LIN {X 0.038,Y -348.064,Z 1859.529,A 0.000,B 0.000,C 90.000,E1 275.163} C_DIS
LIN {X -0.149,Y -343.133,Z 1859.525,A 0.000,B 0.000,C 90.000,E1 274.588} C_DIS
LIN {X 0.037,Y -337.603,Z 1859.522,A 0.000,B 0.000,C 90.000,E1 273.955} C_DIS
LIN {X 0.034,Y -331.682,Z 1859.519,A 0.000,B 0.000,C 90.000,E1 273.383} C_DIS
LIN {X -0.019,Y -325.520,Z 1859.516,A 0.000,B 0.000,C 90.000,E1 272.865} C_DIS
LIN {X -0.139,Y -319.108,Z 1859.513,A 0.000,B 0.000,C 90.000,E1 272.407} C_DIS
LIN {X 0.029,Y -312.422,Z 1859.511,A 0.000,B 0.000,C 90.000,E1 271.949} C_DIS
LIN {X -0.128,Y -305.605,Z 1859.509,A 0.000,B 0.000,C 90.000,E1 271.604} C_DIS
LIN {X 0.010,Y -298.212,Z 1859.507,A 0.000,B 0.000,C 90.000,E1 271.260} C_DIS
LIN {X -0.113,Y -290.603,Z 1859.506,A 0.000,B 0.000,C 90.000,E1 271.031} C_DIS
LIN {X 0.034,Y -283.001,Z 1859.505,A 0.000,B 0.000,C 90.000,E1 270.802} C_DIS
LIN {X -0.029,Y -268.014,Z 1859.503,A 0.000,B 0.000,C 90.000,E1 270.516} C_DIS
LIN {X -0.049,Y -246.564,Z 1859.501,A 0.000,B 0.000,C 90.000,E1 270.115} C_DIS
LIN {X -0.031,Y -234.364,Z 1859.500,A 0.000,B 0.000,C 90.000,E1 269.943} C_DIS
LIN {X 0.025,Y -226.280,Z 1859.499,A 0.000,B 0.000,C 90.000,E1 269.885} C_DIS
LIN {X 0.000,Y -181.539,Z 1859.499,A 0.000,B 0.000,C 90.000,E1 269.885} C_DIS
LIN {X -0.082,Y -180.788,Z 1859.471,A 0.000,B 0.000,C 90.000,E1 264.780} C_DIS
LIN {X -0.008,Y -178.886,Z 1859.443,A 0.000,B 0.000,C 90.000,E1 259.690} C_DIS
LIN {X 0.067,Y -175.929,Z 1859.414,A 0.000,B 0.000,C 90.000,E1 254.574} C_DIS
LIN {X 0.013,Y -175.371,Z 1859.410,A 0.000,B 0.000,C 90.000,E1 253.740} C_DIS
LIN {X 0.072,Y -172.148,Z 1859.386,A 0.000,B 0.000,C 90.000,E1 249.444} C_DIS
LIN {X 0.048,Y -171.613,Z 1859.381,A 0.000,B 0.000,C 90.000,E1 248.592} C_DIS
LIN {X 0.036,Y -167.835,Z 1859.357,A 0.000,B 0.000,C 90.000,E1 244.280} C_DIS
LIN {X 0.054,Y -166.562,Z 1859.348,A 0.000,B 0.000,C 90.000,E1 242.538} C_DIS
LIN {X -0.036,Y -162.556,Z 1859.323,A 0.000,B 0.000,C 90.000,E1 238.201} C_DIS
LIN {X 0.023,Y -161.235,Z 1859.313,A 0.000,B 0.000,C 90.000,E1 236.421} C_DIS
LIN {X 0.058,Y -157.240,Z 1859.289,A 0.000,B 0.000,C 90.000,E1 231.984} C_DIS
LIN {X -0.019,Y -155.963,Z 1859.279,A 0.000,B 0.000,C 90.000,E1 230.231} C_DIS
LIN {X 0.039,Y -152.218,Z 1859.254,A 0.000,B 0.000,C 90.000,E1 225.729} C_DIS
LIN {X 0.060,Y -150.462,Z 1859.239,A 0.000,B 0.000,C 90.000,E1 223.014} C_DIS
LIN {X 0.086,Y -147.187,Z 1859.214,A 0.000,B 0.000,C 90.000,E1 218.463} C_DIS
LIN {X 0.052,Y -145.205,Z 1859.194,A 0.000,B 0.000,C 90.000,E1 214.818} C_DIS
LIN {X -0.038,Y -142.340,Z 1859.163,A 0.000,B 0.000,C 90.000,E1 209.333} C_DIS
LIN {X 0.016,Y -141.729,Z 1859.153,A 0.000,B 0.000,C 90.000,E1 207.462} C_DIS
LIN {X -0.003,Y -139.482,Z 1859.116,A 0.000,B 0.000,C 90.000,E1 200.972} C_DIS
LIN {X -0.014,Y -138.980,Z 1859.101,A 0.000,B 0.000,C 90.000,E1 198.181} C_DIS
LIN {X -0.053,Y -138.332,Z 1859.054,A 0.000,B 0.000,C 90.000,E1 189.792} C_DIS
LIN {X -0.028,Y -139.427,Z 1859.008,A 0.000,B 0.000,C 90.000,E1 181.375} C_DIS
LIN {X 0.025,Y -141.354,Z 1858.971,A 0.000,B 0.000,C 90.000,E1 174.837} C_DIS
LIN {X 0.002,Y -142.707,Z 1858.956,A 0.000,B 0.000,C 90.000,E1 172.064} C_DIS
LIN {X -0.040,Y -145.081,Z 1858.930,A 0.000,B 0.000,C 90.000,E1 167.465} C_DIS
LIN {X -0.044,Y -147.706,Z 1858.910,A 0.000,B 0.000,C 90.000,E1 163.795} C_DIS
LIN {X 0.040,Y -150.359,Z 1858.890,A 0.000,B 0.000,C 90.000,E1 160.115} C_DIS
LIN {X 0.058,Y -153.784,Z 1858.870,A 0.000,B 0.000,C 90.000,E1 156.485} C_DIS
LIN {X -0.021,Y -157.197,Z 1858.849,A 0.000,B 0.000,C 90.000,E1 152.922} C_DIS
LIN {X 0.060,Y -161.358,Z 1858.830,A 0.000,B 0.000,C 90.000,E1 149.331} C_DIS
LIN {X 0.072,Y -165.561,Z 1858.810,A 0.000,B 0.000,C 90.000,E1 145.801} C_DIS
LIN {X -0.044,Y -170.477,Z 1858.791,A 0.000,B 0.000,C 90.000,E1 142.351} C_DIS
LIN {X 0.105,Y -175.358,Z 1858.772,A 0.000,B 0.000,C 90.000,E1 138.852} C_DIS
LIN {X -0.032,Y -180.982,Z 1858.753,A 0.000,B 0.000,C 90.000,E1 135.486} C_DIS
LIN {X -0.045,Y -186.408,Z 1858.734,A 0.000,B 0.000,C 90.000,E1 132.123} C_DIS
LIN {X -0.106,Y -191.036,Z 1858.720,A 0.000,B 0.000,C 90.000,E1 129.644} C_DIS
LIN {X 0.086,Y -196.818,Z 1858.702,A 0.000,B 0.000,C 90.000,E1 126.297} C_DIS
LIN {X 0.005,Y -200.073,Z 1858.693,A 0.000,B 0.000,C 90.000,E1 124.692} C_DIS
LIN {X -0.001,Y -207.572,Z 1858.670,A 0.000,B 0.000,C 90.000,E1 120.669} C_DIS
LIN {X 0.002,Y -210.778,Z 1858.661,A 0.000,B 0.000,C 90.000,E1 119.077} C_DIS
LIN {X 0.010,Y -216.622,Z 1858.644,A 0.000,B 0.000,C 90.000,E1 115.924} C_DIS
LIN {X -0.080,Y -219.706,Z 1858.635,A 0.000,B 0.000,C 90.000,E1 114.387} C_DIS
LIN {X 0.069,Y -224.078,Z 1858.621,A 0.000,B 0.000,C 90.000,E1 111.844} C_DIS
LIN {X 0.051,Y -283.399,Z 1858.621,A 0.000,B 0.000,C 90.000,E1 111.844} C_DIS
LIN {X 0.136,Y -286.194,Z 1858.621,A 0.000,B 0.000,C 90.000,E1 111.770} C_DIS
LIN {X 0.002,Y -290.672,Z 1858.620,A 0.000,B 0.000,C 90.000,E1 111.535} C_DIS
LIN {X -0.029,Y -293.267,Z 1858.618,A 0.000,B 0.000,C 90.000,E1 111.280} C_DIS
LIN {X -0.184,Y -297.015,Z 1858.615,A 0.000,B 0.000,C 90.000,E1 110.737} C_DIS
LIN {X 0.111,Y -310.328,Z 1858.602,A 0.000,B 0.000,C 90.000,E1 108.362} C_DIS
LIN {X -0.076,Y -325.008,Z 1858.590,A 0.000,B 0.000,C 90.000,E1 106.134} C_DIS
LIN {X -0.094,Y -338.778,Z 1858.579,A 0.000,B 0.000,C 90.000,E1 104.245} C_DIS
LIN {X 0.162,Y -353.741,Z 1858.569,A 0.000,B 0.000,C 90.000,E1 102.355} C_DIS
LIN {X -0.081,Y -372.155,Z 1858.557,A 0.000,B 0.000,C 90.000,E1 100.366} C_DIS
LIN {X -0.019,Y -391.045,Z 1858.547,A 0.000,B 0.000,C 90.000,E1 98.511} C_DIS
LIN {X -0.022,Y -410.274,Z 1858.538,A 0.000,B 0.000,C 90.000,E1 96.834} C_DIS
LIN {X -0.127,Y -432.668,Z 1858.528,A 0.000,B 0.000,C 90.000,E1 95.106} C_DIS
LIN {X -0.159,Y -438.325,Z 1858.526,A 0.000,B 0.000,C 90.000,E1 94.702} C_DIS
LIN {X 0.046,Y -440.785,Z 1858.525,A 0.000,B 0.000,C 90.000,E1 94.473} C_DIS
LIN {X 0.181,Y -444.365,Z 1858.522,A 0.000,B 0.000,C 90.000,E1 94.012} C_DIS
LIN {X -0.093,Y -445.799,Z 1858.521,A 0.000,B 0.000,C 90.000,E1 93.784} C_DIS
LIN {X 0.079,Y -446.874,Z 1858.520,A 0.000,B 0.000,C 90.000,E1 93.498} C_DIS
LIN {X 0.033,Y -448.156,Z 1858.517,A 0.000,B 0.000,C 90.000,E1 92.980} C_DIS
LIN {X -0.029,Y -448.461,Z 1858.514,A 0.000,B 0.000,C 90.000,E1 92.465} C_DIS
LIN {X -0.082,Y -447.838,Z 1858.511,A 0.000,B 0.000,C 90.000,E1 91.949} C_DIS
LIN {X -0.118,Y -446.196,Z 1858.508,A 0.000,B 0.000,C 90.000,E1 91.432} C_DIS
LIN {X 0.078,Y -444.907,Z 1858.506,A 0.000,B 0.000,C 90.000,E1 91.146} C_DIS
LIN {X 0.008,Y -433.406,Z 1858.496,A 0.000,B 0.000,C 90.000,E1 89.312} C_DIS
LIN {X 0.020,Y -423.403,Z 1858.487,A 0.000,B 0.000,C 90.000,E1 87.707} C_DIS
LIN {X -0.030,Y -411.622,Z 1858.477,A 0.000,B 0.000,C 90.000,E1 85.812} C_DIS
LIN {X 0.122,Y -399.742,Z 1858.466,A 0.000,B 0.000,C 90.000,E1 83.856} C_DIS
LIN {X 0.057,Y -387.787,Z 1858.455,A 0.000,B 0.000,C 90.000,E1 81.894} C_DIS
LIN {X -0.131,Y -375.877,Z 1858.444,A 0.000,B 0.000,C 90.000,E1 79.916} C_DIS
LIN {X 0.121,Y -357.712,Z 1858.426,A 0.000,B 0.000,C 90.000,E1 76.645} C_DIS
LIN {X 0.086,Y -342.275,Z 1858.409,A 0.000,B 0.000,C 90.000,E1 73.630} C_DIS
LIN {X 0.140,Y -330.364,Z 1858.395,A 0.000,B 0.000,C 90.000,E1 71.148} C_DIS
LIN {X 0.027,Y -318.726,Z 1858.381,A 0.000,B 0.000,C 90.000,E1 68.646} C_DIS
LIN {X 0.063,Y -306.241,Z 1858.365,A 0.000,B 0.000,C 90.000,E1 65.741} C_DIS
LIN {X -0.036,Y -296.668,Z 1858.353,A 0.000,B 0.000,C 90.000,E1 63.461} C_DIS
LIN {X -0.088,Y -285.985,Z 1858.338,A 0.000,B 0.000,C 90.000,E1 60.795} C_DIS
LIN {X -0.072,Y -276.568,Z 1858.324,A 0.000,B 0.000,C 90.000,E1 58.408} C_DIS
LIN {X 0.019,Y -267.105,Z 1858.311,A 0.000,B 0.000,C 90.000,E1 55.960} C_DIS
LIN {X -0.016,Y -257.528,Z 1858.297,A 0.000,B 0.000,C 90.000,E1 53.497} C_DIS
LIN {X 0.042,Y -247.918,Z 1858.283,A 0.000,B 0.000,C 90.000,E1 50.964} C_DIS
LIN {X -0.008,Y -237.078,Z 1858.267,A 0.000,B 0.000,C 90.000,E1 48.038} C_DIS
LIN {X -0.084,Y -225.302,Z 1858.248,A 0.000,B 0.000,C 90.000,E1 44.676} C_DIS
LIN {X -0.007,Y -214.152,Z 1858.229,A 0.000,B 0.000,C 90.000,E1 41.191} C_DIS
LIN {X -0.087,Y -206.142,Z 1858.214,A 0.000,B 0.000,C 90.000,E1 38.463} C_DIS
LIN {X 0.038,Y -197.835,Z 1858.196,A 0.000,B 0.000,C 90.000,E1 35.231} C_DIS
LIN {X -0.051,Y -190.265,Z 1858.178,A 0.000,B 0.000,C 90.000,E1 32.005} C_DIS
LIN {X -0.032,Y -183.427,Z 1858.159,A 0.000,B 0.000,C 90.000,E1 28.693} C_DIS
LIN {X -0.033,Y -177.257,Z 1858.141,A 0.000,B 0.000,C 90.000,E1 25.335} C_DIS
LIN {X 0.065,Y -171.918,Z 1858.122,A 0.000,B 0.000,C 90.000,E1 21.897} C_DIS
LIN {X -0.053,Y -167.341,Z 1858.103,A 0.000,B 0.000,C 90.000,E1 18.489} C_DIS
LIN {X -0.063,Y -163.572,Z 1858.083,A 0.000,B 0.000,C 90.000,E1 15.009} C_DIS
LIN {X 0.033,Y -161.193,Z 1858.069,A 0.000,B 0.000,C 90.000,E1 12.355} C_DIS
LIN {X 0.014,Y -161.371,Z 1858.069,A 0.000,B 0.000,C 90.000,E1 12.355} C_DIS
LIN {X -0.062,Y -168.654,Z 1858.067,A 0.000,B 0.000,C 90.000,E1 12.119} C_DIS
LIN {X -0.066,Y -173.315,Z 1858.066,A 0.000,B 0.000,C 90.000,E1 11.883} C_DIS
LIN {X 0.008,Y -174.617,Z 1858.064,A 0.000,B 0.000,C 90.000,E1 11.535} C_DIS
LIN {X 0.065,Y -176.312,Z 1858.059,A 0.000,B 0.000,C 90.000,E1 10.658} C_DIS
LIN {X -0.076,Y -177.310,Z 1858.055,A 0.000,B 0.000,C 90.000,E1 9.849} C_DIS
LIN {X 0.051,Y -178.596,Z 1858.045,A 0.000,B 0.000,C 90.000,E1 8.106} C_DIS
LIN {X 0.036,Y -179.856,Z 1858.031,A 0.000,B 0.000,C 90.000,E1 5.568} C_DIS
LIN {X 0.071,Y -181.214,Z 1858.012,A 0.000,B 0.000,C 90.000,E1 2.178} C_DIS
LIN {X 0.026,Y -182.550,Z 1857.993,A 0.000,B 0.000,C 90.000,E1 358.682} C_DIS
LIN {X 0.018,Y -184.224,Z 1857.969,A 0.000,B 0.000,C 90.000,E1 354.489} C_DIS
LIN {X -0.049,Y -186.005,Z 1857.946,A 0.000,B 0.000,C 90.000,E1 350.330} C_DIS
LIN {X -0.063,Y -187.969,Z 1857.923,A 0.000,B 0.000,C 90.000,E1 346.172} C_DIS
LIN {X 0.031,Y -190.042,Z 1857.900,A 0.000,B 0.000,C 90.000,E1 342.000} C_DIS
LIN {X -0.052,Y -192.174,Z 1857.877,A 0.000,B 0.000,C 90.000,E1 337.901} C_DIS
LIN {X 0.044,Y -194.600,Z 1857.854,A 0.000,B 0.000,C 90.000,E1 333.768} C_DIS
LIN {X 0.120,Y -197.468,Z 1857.832,A 0.000,B 0.000,C 90.000,E1 329.665} C_DIS
LIN {X -0.100,Y -200.742,Z 1857.809,A 0.000,B 0.000,C 90.000,E1 325.674} C_DIS
LIN {X 0.014,Y -204.489,Z 1857.787,A 0.000,B 0.000,C 90.000,E1 321.618} C_DIS
LIN {X -0.012,Y -208.970,Z 1857.765,A 0.000,B 0.000,C 90.000,E1 317.634} C_DIS
LIN {X 0.044,Y -212.502,Z 1857.751,A 0.000,B 0.000,C 90.000,E1 315.243} C_DIS
LIN {X -0.084,Y -215.374,Z 1857.743,A 0.000,B 0.000,C 90.000,E1 313.704} C_DIS
LIN {X -0.026,Y -218.859,Z 1857.734,A 0.000,B 0.000,C 90.000,E1 312.123} C_DIS
LIN {X 0.032,Y -222.027,Z 1857.728,A 0.000,B 0.000,C 90.000,E1 310.943} C_DIS
LIN {X 0.037,Y -227.047,Z 1857.719,A 0.000,B 0.000,C 90.000,E1 309.402} C_DIS
LIN {X -0.010,Y -232.983,Z 1857.710,A 0.000,B 0.000,C 90.000,E1 307.890} C_DIS
LIN {X -0.010,Y -241.316,Z 1857.700,A 0.000,B 0.000,C 90.000,E1 306.011} C_DIS
LIN {X 0.045,Y -252.464,Z 1857.688,A 0.000,B 0.000,C 90.000,E1 303.785} C_DIS
LIN {X -0.068,Y -262.636,Z 1857.678,A 0.000,B 0.000,C 90.000,E1 302.005} C_DIS
LIN {X 0.104,Y -280.681,Z 1857.662,A 0.000,B 0.000,C 90.000,E1 299.155} C_DIS
LIN {X -0.004,Y -294.750,Z 1857.651,A 0.000,B 0.000,C 90.000,E1 297.129} C_DIS
LIN {X -0.106,Y -311.109,Z 1857.638,A 0.000,B 0.000,C 90.000,E1 294.823} C_DIS
LIN {X -0.115,Y -322.594,Z 1857.629,A 0.000,B 0.000,C 90.000,E1 293.206} C_DIS
LIN {X 0.059,Y -333.985,Z 1857.620,A 0.000,B 0.000,C 90.000,E1 291.589} C_DIS
LIN {X -0.019,Y -342.628,Z 1857.613,A 0.000,B 0.000,C 90.000,E1 290.355} C_DIS
LIN {X -0.125,Y -348.736,Z 1857.608,A 0.000,B 0.000,C 90.000,E1 289.450} C_DIS
LIN {X -0.180,Y -354.367,Z 1857.603,A 0.000,B 0.000,C 90.000,E1 288.544} C_DIS
LIN {X -0.175,Y -359.498,Z 1857.598,A 0.000,B 0.000,C 90.000,E1 287.638} C_DIS
LIN {X -0.183,Y -362.504,Z 1857.594,A 0.000,B 0.000,C 90.000,E1 287.040} C_DIS
LIN {X -0.109,Y -366.336,Z 1857.590,A 0.000,B 0.000,C 90.000,E1 286.134} C_DIS
LIN {X -0.073,Y -368.536,Z 1857.586,A 0.000,B 0.000,C 90.000,E1 285.536} C_DIS
LIN {X -0.119,Y -370.412,Z 1857.583,A 0.000,B 0.000,C 90.000,E1 284.954} C_DIS
LIN {X -0.062,Y -371.957,Z 1857.580,A 0.000,B 0.000,C 90.000,E1 284.356} C_DIS
LIN {X -0.085,Y -373.166,Z 1857.576,A 0.000,B 0.000,C 90.000,E1 283.772} C_DIS
LIN {X -0.009,Y -373.952,Z 1857.573,A 0.000,B 0.000,C 90.000,E1 283.175} C_DIS
LIN {X -0.013,Y -374.290,Z 1857.570,A 0.000,B 0.000,C 90.000,E1 282.591} C_DIS
LIN {X -0.010,Y -374.270,Z 1857.567,A 0.000,B 0.000,C 90.000,E1 282.007} C_DIS
LIN {X -0.004,Y -373.756,Z 1857.563,A 0.000,B 0.000,C 90.000,E1 281.422} C_DIS
LIN {X 0.002,Y -372.797,Z 1857.560,A 0.000,B 0.000,C 90.000,E1 280.838} C_DIS
LIN {X 0.004,Y -371.382,Z 1857.557,A 0.000,B 0.000,C 90.000,E1 280.254} C_DIS
LIN {X -0.001,Y -369.598,Z 1857.554,A 0.000,B 0.000,C 90.000,E1 279.670} C_DIS
LIN {X -0.100,Y -365.296,Z 1857.547,A 0.000,B 0.000,C 90.000,E1 278.511} C_DIS
LIN {X 0.131,Y -361.904,Z 1857.542,A 0.000,B 0.000,C 90.000,E1 277.587} C_DIS
LIN {X -0.024,Y -357.905,Z 1857.537,A 0.000,B 0.000,C 90.000,E1 276.720} C_DIS
LIN {X -0.158,Y -354.621,Z 1857.534,A 0.000,B 0.000,C 90.000,E1 276.144} C_DIS
LIN {X 0.041,Y -350.762,Z 1857.531,A 0.000,B 0.000,C 90.000,E1 275.511} C_DIS
LIN {X -0.129,Y -346.239,Z 1857.527,A 0.000,B 0.000,C 90.000,E1 274.935} C_DIS
LIN {X 0.020,Y -340.995,Z 1857.524,A 0.000,B 0.000,C 90.000,E1 274.302} C_DIS
LIN {X -0.075,Y -335.289,Z 1857.521,A 0.000,B 0.000,C 90.000,E1 273.726} C_DIS
LIN {X 0.038,Y -329.268,Z 1857.518,A 0.000,B 0.000,C 90.000,E1 273.154} C_DIS
LIN {X 0.102,Y -322.974,Z 1857.515,A 0.000,B 0.000,C 90.000,E1 272.636} C_DIS
LIN {X 0.114,Y -316.430,Z 1857.512,A 0.000,B 0.000,C 90.000,E1 272.178} C_DIS
LIN {X 0.108,Y -309.709,Z 1857.510,A 0.000,B 0.000,C 90.000,E1 271.776} C_DIS
LIN {X 0.073,Y -302.777,Z 1857.508,A 0.000,B 0.000,C 90.000,E1 271.432} C_DIS
LIN {X 0.018,Y -294.936,Z 1857.506,A 0.000,B 0.000,C 90.000,E1 271.146} C_DIS
LIN {X 0.048,Y -287.555,Z 1857.505,A 0.000,B 0.000,C 90.000,E1 270.917} C_DIS
LIN {X -0.071,Y -276.389,Z 1857.504,A 0.000,B 0.000,C 90.000,E1 270.688} C_DIS
LIN {X 0.070,Y -247.788,Z 1857.501,A 0.000,B 0.000,C 90.000,E1 270.115} C_DIS
LIN {X -0.024,Y -238.998,Z 1857.500,A 0.000,B 0.000,C 90.000,E1 270.000} C_DIS
LIN {X 0.067,Y -225.861,Z 1857.500,A 0.000,B 0.000,C 90.000,E1 269.885} C_DIS
LIN {X 0.033,Y -181.541,Z 1857.499,A 0.000,B 0.000,C 90.000,E1 269.885} C_DIS
LIN {X -0.030,Y -180.795,Z 1857.471,A 0.000,B 0.000,C 90.000,E1 264.780} C_DIS
LIN {X 0.044,Y -178.894,Z 1857.443,A 0.000,B 0.000,C 90.000,E1 259.690} C_DIS
LIN {X -0.050,Y -175.936,Z 1857.415,A 0.000,B 0.000,C 90.000,E1 254.629} C_DIS
LIN {X 0.065,Y -175.386,Z 1857.410,A 0.000,B 0.000,C 90.000,E1 253.740} C_DIS
LIN {X -0.099,Y -172.157,Z 1857.386,A 0.000,B 0.000,C 90.000,E1 249.518} C_DIS
LIN {X -0.061,Y -171.625,Z 1857.381,A 0.000,B 0.000,C 90.000,E1 248.646} C_DIS
LIN {X 0.087,Y -167.848,Z 1857.357,A 0.000,B 0.000,C 90.000,E1 244.280} C_DIS
LIN {X 0.027,Y -166.578,Z 1857.348,A 0.000,B 0.000,C 90.000,E1 242.564} C_DIS
LIN {X 0.012,Y -162.570,Z 1857.323,A 0.000,B 0.000,C 90.000,E1 238.201} C_DIS
LIN {X 0.072,Y -161.251,Z 1857.314,A 0.000,B 0.000,C 90.000,E1 236.421} C_DIS
LIN {X -0.018,Y -157.253,Z 1857.289,A 0.000,B 0.000,C 90.000,E1 232.029} C_DIS
LIN {X 0.029,Y -155.975,Z 1857.279,A 0.000,B 0.000,C 90.000,E1 230.231} C_DIS
LIN {X 0.086,Y -152.231,Z 1857.254,A 0.000,B 0.000,C 90.000,E1 225.729} C_DIS
LIN {X -0.003,Y -150.473,Z 1857.239,A 0.000,B 0.000,C 90.000,E1 223.056} C_DIS
LIN {X -0.074,Y -147.198,Z 1857.214,A 0.000,B 0.000,C 90.000,E1 218.543} C_DIS
LIN {X -0.021,Y -145.217,Z 1857.194,A 0.000,B 0.000,C 90.000,E1 214.865} C_DIS
LIN {X 0.008,Y -142.347,Z 1857.163,A 0.000,B 0.000,C 90.000,E1 209.333} C_DIS
LIN {X -0.065,Y -141.735,Z 1857.153,A 0.000,B 0.000,C 90.000,E1 207.513} C_DIS
LIN {X 0.042,Y -139.485,Z 1857.117,A 0.000,B 0.000,C 90.000,E1 200.972} C_DIS
LIN {X 0.031,Y -138.986,Z 1857.101,A 0.000,B 0.000,C 90.000,E1 198.181} C_DIS
LIN {X -0.008,Y -138.334,Z 1857.054,A 0.000,B 0.000,C 90.000,E1 189.792} C_DIS
LIN {X 0.016,Y -139.424,Z 1857.008,A 0.000,B 0.000,C 90.000,E1 181.375} C_DIS
LIN {X -0.070,Y -141.345,Z 1856.971,A 0.000,B 0.000,C 90.000,E1 174.894} C_DIS
LIN {X 0.047,Y -142.700,Z 1856.956,A 0.000,B 0.000,C 90.000,E1 172.064} C_DIS
LIN {X 0.007,Y -145.070,Z 1856.930,A 0.000,B 0.000,C 90.000,E1 167.465} C_DIS
LIN {X 0.002,Y -147.694,Z 1856.910,A 0.000,B 0.000,C 90.000,E1 163.795} C_DIS
LIN {X 0.036,Y -150.345,Z 1856.890,A 0.000,B 0.000,C 90.000,E1 160.134} C_DIS
LIN {X 0.029,Y -154.599,Z 1856.865,A 0.000,B 0.000,C 90.000,E1 155.613} C_DIS
LIN {X 0.036,Y -158.139,Z 1856.845,A 0.000,B 0.000,C 90.000,E1 152.025} C_DIS
LIN {X -0.004,Y -162.426,Z 1856.825,A 0.000,B 0.000,C 90.000,E1 148.486} C_DIS
LIN {X -0.023,Y -166.683,Z 1856.805,A 0.000,B 0.000,C 90.000,E1 144.975} C_DIS
LIN {X 0.090,Y -171.689,Z 1856.786,A 0.000,B 0.000,C 90.000,E1 141.457} C_DIS
LIN {X 0.025,Y -176.660,Z 1856.767,A 0.000,B 0.000,C 90.000,E1 138.038} C_DIS
LIN {X 0.021,Y -180.957,Z 1856.753,A 0.000,B 0.000,C 90.000,E1 135.486} C_DIS
LIN {X 0.008,Y -186.379,Z 1856.734,A 0.000,B 0.000,C 90.000,E1 132.123} C_DIS
LIN {X -0.051,Y -191.009,Z 1856.720,A 0.000,B 0.000,C 90.000,E1 129.644} C_DIS
LIN {X -0.017,Y -196.787,Z 1856.702,A 0.000,B 0.000,C 90.000,E1 126.343} C_DIS
LIN {X 0.061,Y -200.039,Z 1856.693,A 0.000,B 0.000,C 90.000,E1 124.692} C_DIS
LIN {X 0.055,Y -207.540,Z 1856.670,A 0.000,B 0.000,C 90.000,E1 120.669} C_DIS
LIN {X 0.060,Y -210.752,Z 1856.662,A 0.000,B 0.000,C 90.000,E1 119.077} C_DIS
LIN {X 0.068,Y -216.592,Z 1856.644,A 0.000,B 0.000,C 90.000,E1 115.924} C_DIS
LIN {X -0.021,Y -219.681,Z 1856.635,A 0.000,B 0.000,C 90.000,E1 114.387} C_DIS
LIN {X 0.071,Y -224.077,Z 1856.621,A 0.000,B 0.000,C 90.000,E1 111.844} C_DIS
LIN {X 0.059,Y -283.411,Z 1856.621,A 0.000,B 0.000,C 90.000,E1 111.844} C_DIS
LIN {X -0.161,Y -285.776,Z 1856.621,A 0.000,B 0.000,C 90.000,E1 111.844} C_DIS
LIN {X 0.078,Y -290.500,Z 1856.620,A 0.000,B 0.000,C 90.000,E1 111.535} C_DIS
LIN {X 0.048,Y -293.143,Z 1856.618,A 0.000,B 0.000,C 90.000,E1 111.280} C_DIS
LIN {X -0.062,Y -296.887,Z 1856.615,A 0.000,B 0.000,C 90.000,E1 110.737} C_DIS
LIN {X -0.059,Y -310.186,Z 1856.602,A 0.000,B 0.000,C 90.000,E1 108.417} C_DIS
LIN {X 0.051,Y -324.852,Z 1856.590,A 0.000,B 0.000,C 90.000,E1 106.134} C_DIS
LIN {X 0.035,Y -338.609,Z 1856.579,A 0.000,B 0.000,C 90.000,E1 104.245} C_DIS
LIN {X -0.052,Y -353.557,Z 1856.569,A 0.000,B 0.000,C 90.000,E1 102.411} C_DIS
LIN {X 0.045,Y -371.967,Z 1856.558,A 0.000,B 0.000,C 90.000,E1 100.366} C_DIS
LIN {X 0.102,Y -390.851,Z 1856.547,A 0.000,B 0.000,C 90.000,E1 98.511} C_DIS
LIN {X 0.092,Y -410.078,Z 1856.538,A 0.000,B 0.000,C 90.000,E1 96.834} C_DIS
LIN {X -0.018,Y -432.469,Z 1856.528,A 0.000,B 0.000,C 90.000,E1 95.106} C_DIS
LIN {X -0.051,Y -438.125,Z 1856.526,A 0.000,B 0.000,C 90.000,E1 94.702} C_DIS
LIN {X 0.153,Y -440.633,Z 1856.525,A 0.000,B 0.000,C 90.000,E1 94.473} C_DIS
LIN {X -0.141,Y -444.231,Z 1856.523,A 0.000,B 0.000,C 90.000,E1 94.073} C_DIS
LIN {X 0.061,Y -445.695,Z 1856.521,A 0.000,B 0.000,C 90.000,E1 93.784} C_DIS
LIN {X -0.214,Y -446.793,Z 1856.520,A 0.000,B 0.000,C 90.000,E1 93.555} C_DIS
LIN {X 0.187,Y -448.114,Z 1856.517,A 0.000,B 0.000,C 90.000,E1 92.980} C_DIS
LIN {X 0.123,Y -448.451,Z 1856.514,A 0.000,B 0.000,C 90.000,E1 92.465} C_DIS
LIN {X 0.070,Y -447.863,Z 1856.511,A 0.000,B 0.000,C 90.000,E1 91.949} C_DIS
LIN {X 0.033,Y -446.261,Z 1856.508,A 0.000,B 0.000,C 90.000,E1 91.432} C_DIS
LIN {X -0.216,Y -444.997,Z 1856.506,A 0.000,B 0.000,C 90.000,E1 91.203} C_DIS
LIN {X 0.157,Y -433.508,Z 1856.496,A 0.000,B 0.000,C 90.000,E1 89.312} C_DIS
LIN {X 0.167,Y -423.510,Z 1856.487,A 0.000,B 0.000,C 90.000,E1 87.707} C_DIS
LIN {X 0.115,Y -411.728,Z 1856.477,A 0.000,B 0.000,C 90.000,E1 85.812} C_DIS
LIN {X -0.132,Y -399.849,Z 1856.466,A 0.000,B 0.000,C 90.000,E1 83.913} C_DIS
LIN {X -0.185,Y -387.895,Z 1856.455,A 0.000,B 0.000,C 90.000,E1 81.951} C_DIS
LIN {X -0.057,Y -375.983,Z 1856.444,A 0.000,B 0.000,C 90.000,E1 79.926} C_DIS
LIN {X -0.054,Y -359.403,Z 1856.428,A 0.000,B 0.000,C 90.000,E1 76.992} C_DIS
LIN {X -0.022,Y -343.878,Z 1856.411,A 0.000,B 0.000,C 90.000,E1 73.976} C_DIS
LIN {X -0.020,Y -331.934,Z 1856.397,A 0.000,B 0.000,C 90.000,E1 71.511} C_DIS
LIN {X 0.095,Y -320.246,Z 1856.383,A 0.000,B 0.000,C 90.000,E1 68.975} C_DIS
LIN {X -0.004,Y -307.673,Z 1856.367,A 0.000,B 0.000,C 90.000,E1 66.102} C_DIS
LIN {X -0.076,Y -299.486,Z 1856.356,A 0.000,B 0.000,C 90.000,E1 64.152} C_DIS
LIN {X 0.052,Y -287.398,Z 1856.340,A 0.000,B 0.000,C 90.000,E1 61.129} C_DIS
LIN {X 0.089,Y -277.988,Z 1856.326,A 0.000,B 0.000,C 90.000,E1 58.742} C_DIS
LIN {X -0.011,Y -268.534,Z 1856.313,A 0.000,B 0.000,C 90.000,E1 56.342} C_DIS
LIN {X 0.150,Y -260.345,Z 1856.301,A 0.000,B 0.000,C 90.000,E1 54.196} C_DIS
LIN {X -0.084,Y -250.739,Z 1856.287,A 0.000,B 0.000,C 90.000,E1 51.743} C_DIS
LIN {X -0.014,Y -241.197,Z 1856.273,A 0.000,B 0.000,C 90.000,E1 49.175} C_DIS
LIN {X -0.085,Y -230.505,Z 1856.257,A 0.000,B 0.000,C 90.000,E1 46.215} C_DIS
LIN {X 0.057,Y -220.320,Z 1856.240,A 0.000,B 0.000,C 90.000,E1 43.137} C_DIS
LIN {X 0.121,Y -210.704,Z 1856.222,A 0.000,B 0.000,C 90.000,E1 40.011} C_DIS
LIN {X 0.017,Y -201.945,Z 1856.205,A 0.000,B 0.000,C 90.000,E1 36.870} C_DIS
LIN {X -0.023,Y -194.018,Z 1856.187,A 0.000,B 0.000,C 90.000,E1 33.658} C_DIS
LIN {X -0.041,Y -186.819,Z 1856.169,A 0.000,B 0.000,C 90.000,E1 30.384} C_DIS
LIN {X -0.041,Y -180.301,Z 1856.150,A 0.000,B 0.000,C 90.000,E1 27.052} C_DIS
LIN {X -0.027,Y -175.883,Z 1856.136,A 0.000,B 0.000,C 90.000,E1 24.515} C_DIS
LIN {X -0.028,Y -170.746,Z 1856.117,A 0.000,B 0.000,C 90.000,E1 21.099} C_DIS
LIN {X -0.014,Y -166.357,Z 1856.098,A 0.000,B 0.000,C 90.000,E1 17.638} C_DIS
LIN {X 0.019,Y -164.432,Z 1856.088,A 0.000,B 0.000,C 90.000,E1 15.843} C_DIS
LIN {X 0.000,Y -164.472,Z 1856.088,A 0.000,B 0.000,C 90.000,E1 15.843} C_DIS
LIN {X 0.082,Y -171.691,Z 1856.086,A 0.000,B 0.000,C 90.000,E1 15.426} C_DIS
LIN {X 0.023,Y -176.651,Z 1856.083,A 0.000,B 0.000,C 90.000,E1 15.009} C_DIS
LIN {X -0.029,Y -178.029,Z 1856.080,A 0.000,B 0.000,C 90.000,E1 14.481} C_DIS
LIN {X 0.091,Y -179.183,Z 1856.076,A 0.000,B 0.000,C 90.000,E1 13.592} C_DIS
LIN {X 0.003,Y -179.907,Z 1856.071,A 0.000,B 0.000,C 90.000,E1 12.771} C_DIS
LIN {X 0.022,Y -180.803,Z 1856.062,A 0.000,B 0.000,C 90.000,E1 11.074} C_DIS
LIN {X -0.052,Y -181.575,Z 1856.047,A 0.000,B 0.000,C 90.000,E1 8.568} C_DIS
LIN {X 0.070,Y -182.277,Z 1856.029,A 0.000,B 0.000,C 90.000,E1 5.163} C_DIS
LIN {X 0.037,Y -183.248,Z 1856.005,A 0.000,B 0.000,C 90.000,E1 0.974} C_DIS
LIN {X -0.006,Y -184.331,Z 1855.983,A 0.000,B 0.000,C 90.000,E1 357.020} C_DIS
LIN {X -0.036,Y -185.430,Z 1855.965,A 0.000,B 0.000,C 90.000,E1 353.685} C_DIS
LIN {X -0.018,Y -186.932,Z 1855.942,A 0.000,B 0.000,C 90.000,E1 349.511} C_DIS
LIN {X 0.028,Y -188.303,Z 1855.923,A 0.000,B 0.000,C 90.000,E1 346.172} C_DIS
LIN {X -0.048,Y -190.119,Z 1855.900,A 0.000,B 0.000,C 90.000,E1 342.054} C_DIS
LIN {X -0.020,Y -192.000,Z 1855.877,A 0.000,B 0.000,C 90.000,E1 337.922} C_DIS
LIN {X -0.027,Y -194.871,Z 1855.850,A 0.000,B 0.000,C 90.000,E1 332.999} C_DIS
LIN {X -0.019,Y -197.823,Z 1855.827,A 0.000,B 0.000,C 90.000,E1 328.918} C_DIS
LIN {X 0.047,Y -201.215,Z 1855.805,A 0.000,B 0.000,C 90.000,E1 324.848} C_DIS
LIN {X -0.021,Y -205.085,Z 1855.782,A 0.000,B 0.000,C 90.000,E1 320.848} C_DIS
LIN {X -0.023,Y -209.907,Z 1855.760,A 0.000,B 0.000,C 90.000,E1 316.863} C_DIS
LIN {X -0.102,Y -213.763,Z 1855.747,A 0.000,B 0.000,C 90.000,E1 314.514} C_DIS
LIN {X -0.062,Y -216.963,Z 1855.738,A 0.000,B 0.000,C 90.000,E1 312.933} C_DIS
LIN {X 0.015,Y -220.876,Z 1855.730,A 0.000,B 0.000,C 90.000,E1 311.353} C_DIS
LIN {X 0.101,Y -224.412,Z 1855.723,A 0.000,B 0.000,C 90.000,E1 310.172} C_DIS
LIN {X 0.045,Y -228.475,Z 1855.717,A 0.000,B 0.000,C 90.000,E1 309.036} C_DIS
LIN {X 0.016,Y -234.624,Z 1855.708,A 0.000,B 0.000,C 90.000,E1 307.523} C_DIS
LIN {X 0.047,Y -243.165,Z 1855.698,A 0.000,B 0.000,C 90.000,E1 305.644} C_DIS
LIN {X 0.009,Y -256.521,Z 1855.684,A 0.000,B 0.000,C 90.000,E1 303.086} C_DIS
LIN {X 0.085,Y -269.346,Z 1855.672,A 0.000,B 0.000,C 90.000,E1 300.924} C_DIS
LIN {X 0.103,Y -285.540,Z 1855.658,A 0.000,B 0.000,C 90.000,E1 298.487} C_DIS
LIN {X -0.049,Y -297.300,Z 1855.649,A 0.000,B 0.000,C 90.000,E1 296.821} C_DIS
LIN {X 0.012,Y -311.385,Z 1855.638,A 0.000,B 0.000,C 90.000,E1 294.823} C_DIS
LIN {X -0.056,Y -325.251,Z 1855.627,A 0.000,B 0.000,C 90.000,E1 292.898} C_DIS
LIN {X 0.194,Y -334.362,Z 1855.620,A 0.000,B 0.000,C 90.000,E1 291.589} C_DIS
LIN {X 0.006,Y -343.050,Z 1855.613,A 0.000,B 0.000,C 90.000,E1 290.375} C_DIS
LIN {X 0.025,Y -349.176,Z 1855.608,A 0.000,B 0.000,C 90.000,E1 289.450} C_DIS
LIN {X -0.023,Y -354.863,Z 1855.603,A 0.000,B 0.000,C 90.000,E1 288.544} C_DIS
LIN {X -0.012,Y -360.047,Z 1855.598,A 0.000,B 0.000,C 90.000,E1 287.638} C_DIS
LIN {X 0.041,Y -364.384,Z 1855.593,A 0.000,B 0.000,C 90.000,E1 286.732} C_DIS
LIN {X 0.036,Y -368.002,Z 1855.588,A 0.000,B 0.000,C 90.000,E1 285.843} C_DIS
LIN {X 0.065,Y -370.946,Z 1855.583,A 0.000,B 0.000,C 90.000,E1 284.954} C_DIS
LIN {X 0.126,Y -372.482,Z 1855.580,A 0.000,B 0.000,C 90.000,E1 284.356} C_DIS
LIN {X 0.108,Y -373.679,Z 1855.577,A 0.000,B 0.000,C 90.000,E1 283.772} C_DIS
LIN {X 0.187,Y -374.450,Z 1855.573,A 0.000,B 0.000,C 90.000,E1 283.175} C_DIS
LIN {X 0.186,Y -374.830,Z 1855.570,A 0.000,B 0.000,C 90.000,E1 282.591} C_DIS
LIN {X -0.174,Y -374.750,Z 1855.567,A 0.000,B 0.000,C 90.000,E1 282.063} C_DIS
LIN {X -0.166,Y -374.215,Z 1855.564,A 0.000,B 0.000,C 90.000,E1 281.478} C_DIS
LIN {X -0.158,Y -373.263,Z 1855.560,A 0.000,B 0.000,C 90.000,E1 280.894} C_DIS
LIN {X -0.152,Y -371.854,Z 1855.557,A 0.000,B 0.000,C 90.000,E1 280.310} C_DIS
LIN {X -0.154,Y -370.017,Z 1855.554,A 0.000,B 0.000,C 90.000,E1 279.726} C_DIS
LIN {X 0.114,Y -365.622,Z 1855.547,A 0.000,B 0.000,C 90.000,E1 278.511} C_DIS
LIN {X -0.044,Y -360.982,Z 1855.541,A 0.000,B 0.000,C 90.000,E1 277.352} C_DIS
LIN {X -0.164,Y -358.274,Z 1855.537,A 0.000,B 0.000,C 90.000,E1 276.777} C_DIS
LIN {X 0.057,Y -355.072,Z 1855.534,A 0.000,B 0.000,C 90.000,E1 276.144} C_DIS
LIN {X -0.093,Y -351.234,Z 1855.531,A 0.000,B 0.000,C 90.000,E1 275.568} C_DIS
LIN {X 0.086,Y -346.774,Z 1855.527,A 0.000,B 0.000,C 90.000,E1 274.935} C_DIS
LIN {X -0.106,Y -341.540,Z 1855.524,A 0.000,B 0.000,C 90.000,E1 274.359} C_DIS
LIN {X 0.090,Y -335.746,Z 1855.521,A 0.000,B 0.000,C 90.000,E1 273.726} C_DIS
LIN {X -0.146,Y -329.727,Z 1855.518,A 0.000,B 0.000,C 90.000,E1 273.212} C_DIS
LIN {X -0.105,Y -323.325,Z 1855.515,A 0.000,B 0.000,C 90.000,E1 272.694} C_DIS
LIN {X -0.086,Y -316.838,Z 1855.512,A 0.000,B 0.000,C 90.000,E1 272.236} C_DIS
LIN {X -0.087,Y -310.162,Z 1855.510,A 0.000,B 0.000,C 90.000,E1 271.835} C_DIS
LIN {X -0.120,Y -303.168,Z 1855.508,A 0.000,B 0.000,C 90.000,E1 271.489} C_DIS
LIN {X -0.142,Y -295.712,Z 1855.507,A 0.000,B 0.000,C 90.000,E1 271.203} C_DIS
LIN {X 0.128,Y -288.034,Z 1855.505,A 0.000,B 0.000,C 90.000,E1 270.917} C_DIS
LIN {X -0.008,Y -276.738,Z 1855.504,A 0.000,B 0.000,C 90.000,E1 270.688} C_DIS
LIN {X 0.124,Y -248.199,Z 1855.501,A 0.000,B 0.000,C 90.000,E1 270.115} C_DIS
LIN {X 0.036,Y -239.705,Z 1855.500,A 0.000,B 0.000,C 90.000,E1 270.000} C_DIS
LIN {X -0.106,Y -227.959,Z 1855.500,A 0.000,B 0.000,C 90.000,E1 269.943} C_DIS
LIN {X 0.076,Y -181.544,Z 1855.500,A 0.000,B 0.000,C 90.000,E1 269.885} C_DIS
LIN {X 0.006,Y -180.798,Z 1855.471,A 0.000,B 0.000,C 90.000,E1 264.780} C_DIS
LIN {X 0.080,Y -178.898,Z 1855.443,A 0.000,B 0.000,C 90.000,E1 259.690} C_DIS
LIN {X -0.015,Y -175.941,Z 1855.415,A 0.000,B 0.000,C 90.000,E1 254.629} C_DIS
LIN {X -0.068,Y -175.397,Z 1855.410,A 0.000,B 0.000,C 90.000,E1 253.795} C_DIS
LIN {X -0.065,Y -172.165,Z 1855.386,A 0.000,B 0.000,C 90.000,E1 249.518} C_DIS
LIN {X -0.026,Y -171.634,Z 1855.381,A 0.000,B 0.000,C 90.000,E1 248.646} C_DIS
LIN {X -0.030,Y -167.857,Z 1855.357,A 0.000,B 0.000,C 90.000,E1 244.332} C_DIS
LIN {X -0.087,Y -166.588,Z 1855.348,A 0.000,B 0.000,C 90.000,E1 242.615} C_DIS
LIN {X 0.046,Y -162.579,Z 1855.323,A 0.000,B 0.000,C 90.000,E1 238.201} C_DIS
LIN {X 0.107,Y -161.261,Z 1855.314,A 0.000,B 0.000,C 90.000,E1 236.421} C_DIS
LIN {X 0.015,Y -157.263,Z 1855.289,A 0.000,B 0.000,C 90.000,E1 232.029} C_DIS
LIN {X -0.058,Y -155.983,Z 1855.279,A 0.000,B 0.000,C 90.000,E1 230.275} C_DIS
LIN {X -0.097,Y -152.240,Z 1855.254,A 0.000,B 0.000,C 90.000,E1 225.810} C_DIS
LIN {X 0.029,Y -150.481,Z 1855.239,A 0.000,B 0.000,C 90.000,E1 223.056} C_DIS
LIN {X -0.043,Y -147.205,Z 1855.214,A 0.000,B 0.000,C 90.000,E1 218.543} C_DIS
LIN {X -0.072,Y -145.225,Z 1855.194,A 0.000,B 0.000,C 90.000,E1 214.898} C_DIS
LIN {X 0.038,Y -142.352,Z 1855.163,A 0.000,B 0.000,C 90.000,E1 209.333} C_DIS
LIN {X -0.034,Y -141.739,Z 1855.153,A 0.000,B 0.000,C 90.000,E1 207.513} C_DIS
LIN {X 0.072,Y -139.487,Z 1855.117,A 0.000,B 0.000,C 90.000,E1 200.972} C_DIS
LIN {X 0.061,Y -138.989,Z 1855.101,A 0.000,B 0.000,C 90.000,E1 198.181} C_DIS
LIN {X 0.022,Y -138.335,Z 1855.054,A 0.000,B 0.000,C 90.000,E1 189.792} C_DIS
LIN {X 0.047,Y -139.420,Z 1855.008,A 0.000,B 0.000,C 90.000,E1 181.375} C_DIS
LIN {X -0.040,Y -141.339,Z 1854.972,A 0.000,B 0.000,C 90.000,E1 174.894} C_DIS
LIN {X 0.078,Y -142.696,Z 1854.956,A 0.000,B 0.000,C 90.000,E1 172.064} C_DIS
LIN {X 0.038,Y -145.062,Z 1854.930,A 0.000,B 0.000,C 90.000,E1 167.465} C_DIS
LIN {X 0.035,Y -147.687,Z 1854.910,A 0.000,B 0.000,C 90.000,E1 163.795} C_DIS
LIN {X -0.073,Y -150.334,Z 1854.890,A 0.000,B 0.000,C 90.000,E1 160.188} C_DIS
LIN {X -0.002,Y -153.752,Z 1854.870,A 0.000,B 0.000,C 90.000,E1 156.538} C_DIS
LIN {X -0.011,Y -157.166,Z 1854.850,A 0.000,B 0.000,C 90.000,E1 152.948} C_DIS
LIN {X -0.078,Y -161.320,Z 1854.830,A 0.000,B 0.000,C 90.000,E1 149.410} C_DIS
LIN {X 0.076,Y -164.434,Z 1854.815,A 0.000,B 0.000,C 90.000,E1 146.707} C_DIS
LIN {X 0.070,Y -169.120,Z 1854.796,A 0.000,B 0.000,C 90.000,E1 143.210} C_DIS
LIN {X 0.018,Y -171.673,Z 1854.786,A 0.000,B 0.000,C 90.000,E1 141.492} C_DIS
LIN {X -0.070,Y -176.641,Z 1854.767,A 0.000,B 0.000,C 90.000,E1 138.081} C_DIS
LIN {X 0.057,Y -180.939,Z 1854.753,A 0.000,B 0.000,C 90.000,E1 135.486} C_DIS
LIN {X 0.045,Y -186.359,Z 1854.734,A 0.000,B 0.000,C 90.000,E1 132.123} C_DIS
LIN {X -0.014,Y -190.990,Z 1854.720,A 0.000,B 0.000,C 90.000,E1 129.644} C_DIS
LIN {X -0.095,Y -196.766,Z 1854.702,A 0.000,B 0.000,C 90.000,E1 126.377} C_DIS
LIN {X -0.066,Y -200.016,Z 1854.693,A 0.000,B 0.000,C 90.000,E1 124.739} C_DIS
LIN {X 0.095,Y -207.518,Z 1854.671,A 0.000,B 0.000,C 90.000,E1 120.669} C_DIS
LIN {X 0.098,Y -210.734,Z 1854.662,A 0.000,B 0.000,C 90.000,E1 119.077} C_DIS
LIN {X -0.087,Y -216.570,Z 1854.644,A 0.000,B 0.000,C 90.000,E1 115.976} C_DIS
LIN {X 0.019,Y -219.664,Z 1854.635,A 0.000,B 0.000,C 90.000,E1 114.387} C_DIS
LIN {X 0.086,Y -224.069,Z 1854.621,A 0.000,B 0.000,C 90.000,E1 111.844} C_DIS
LIN {X 0.079,Y -282.868,Z 1854.621,A 0.000,B 0.000,C 90.000,E1 111.844} C_DIS
LIN {X -0.109,Y -285.469,Z 1854.621,A 0.000,B 0.000,C 90.000,E1 111.844} C_DIS
LIN {X 0.130,Y -290.382,Z 1854.620,A 0.000,B 0.000,C 90.000,E1 111.535} C_DIS
LIN {X 0.102,Y -293.058,Z 1854.618,A 0.000,B 0.000,C 90.000,E1 111.280} C_DIS
LIN {X 0.020,Y -296.799,Z 1854.615,A 0.000,B 0.000,C 90.000,E1 110.737} C_DIS
LIN {X 0.025,Y -310.091,Z 1854.602,A 0.000,B 0.000,C 90.000,E1 108.417} C_DIS
LIN {X 0.047,Y -324.747,Z 1854.590,A 0.000,B 0.000,C 90.000,E1 106.150} C_DIS
LIN {X 0.123,Y -338.494,Z 1854.579,A 0.000,B 0.000,C 90.000,E1 104.245} C_DIS
LIN {X 0.038,Y -353.432,Z 1854.569,A 0.000,B 0.000,C 90.000,E1 102.411} C_DIS
LIN {X 0.129,Y -371.839,Z 1854.558,A 0.000,B 0.000,C 90.000,E1 100.366} C_DIS
LIN {X 0.182,Y -390.722,Z 1854.547,A 0.000,B 0.000,C 90.000,E1 98.511} C_DIS
LIN {X 0.170,Y -409.946,Z 1854.538,A 0.000,B 0.000,C 90.000,E1 96.834} C_DIS
LIN {X 0.055,Y -432.335,Z 1854.528,A 0.000,B 0.000,C 90.000,E1 95.106} C_DIS
LIN {X 0.021,Y -437.991,Z 1854.526,A 0.000,B 0.000,C 90.000,E1 94.702} C_DIS
LIN {X -0.214,Y -440.529,Z 1854.525,A 0.000,B 0.000,C 90.000,E1 94.531} C_DIS
LIN {X -0.041,Y -444.140,Z 1854.523,A 0.000,B 0.000,C 90.000,E1 94.073} C_DIS
LIN {X 0.161,Y -445.623,Z 1854.521,A 0.000,B 0.000,C 90.000,E1 93.784} C_DIS
LIN {X -0.114,Y -446.737,Z 1854.520,A 0.000,B 0.000,C 90.000,E1 93.555} C_DIS
LIN {X -0.161,Y -448.081,Z 1854.517,A 0.000,B 0.000,C 90.000,E1 93.037} C_DIS
LIN {X 0.223,Y -448.439,Z 1854.514,A 0.000,B 0.000,C 90.000,E1 92.465} C_DIS
LIN {X 0.170,Y -447.873,Z 1854.511,A 0.000,B 0.000,C 90.000,E1 91.949} C_DIS
LIN {X 0.132,Y -446.297,Z 1854.508,A 0.000,B 0.000,C 90.000,E1 91.432} C_DIS
LIN {X -0.117,Y -445.049,Z 1854.507,A 0.000,B 0.000,C 90.000,E1 91.203} C_DIS
LIN {X -0.179,Y -433.568,Z 1854.496,A 0.000,B 0.000,C 90.000,E1 89.370} C_DIS
LIN {X -0.160,Y -423.575,Z 1854.487,A 0.000,B 0.000,C 90.000,E1 87.764} C_DIS
LIN {X 0.210,Y -411.791,Z 1854.477,A 0.000,B 0.000,C 90.000,E1 85.812} C_DIS
LIN {X -0.039,Y -399.913,Z 1854.466,A 0.000,B 0.000,C 90.000,E1 83.913} C_DIS
LIN {X -0.094,Y -387.959,Z 1854.455,A 0.000,B 0.000,C 90.000,E1 81.951} C_DIS
LIN {X 0.033,Y -376.045,Z 1854.444,A 0.000,B 0.000,C 90.000,E1 79.926} C_DIS
LIN {X 0.034,Y -359.460,Z 1854.428,A 0.000,B 0.000,C 90.000,E1 76.992} C_DIS
LIN {X 0.063,Y -343.930,Z 1854.411,A 0.000,B 0.000,C 90.000,E1 73.976} C_DIS
LIN {X 0.064,Y -331.984,Z 1854.397,A 0.000,B 0.000,C 90.000,E1 71.511} C_DIS
LIN {X -0.122,Y -320.291,Z 1854.383,A 0.000,B 0.000,C 90.000,E1 69.028} C_DIS
LIN {X 0.077,Y -307.716,Z 1854.367,A 0.000,B 0.000,C 90.000,E1 66.102} C_DIS
LIN {X 0.021,Y -298.149,Z 1854.355,A 0.000,B 0.000,C 90.000,E1 63.819} C_DIS
LIN {X -0.123,Y -287.436,Z 1854.340,A 0.000,B 0.000,C 90.000,E1 61.179} C_DIS
LIN {X -0.073,Y -278.028,Z 1854.327,A 0.000,B 0.000,C 90.000,E1 58.791} C_DIS
LIN {X 0.061,Y -268.574,Z 1854.313,A 0.000,B 0.000,C 90.000,E1 56.342} C_DIS
LIN {X -0.141,Y -260.387,Z 1854.301,A 0.000,B 0.000,C 90.000,E1 54.276} C_DIS
LIN {X -0.013,Y -250.783,Z 1854.287,A 0.000,B 0.000,C 90.000,E1 51.743} C_DIS
LIN {X 0.055,Y -241.240,Z 1854.273,A 0.000,B 0.000,C 90.000,E1 49.175} C_DIS
LIN {X -0.018,Y -230.546,Z 1854.257,A 0.000,B 0.000,C 90.000,E1 46.215} C_DIS
LIN {X -0.029,Y -220.359,Z 1854.240,A 0.000,B 0.000,C 90.000,E1 43.176} C_DIS
LIN {X -0.114,Y -210.739,Z 1854.223,A 0.000,B 0.000,C 90.000,E1 40.092} C_DIS
LIN {X 0.078,Y -201.977,Z 1854.205,A 0.000,B 0.000,C 90.000,E1 36.870} C_DIS
LIN {X 0.037,Y -194.049,Z 1854.187,A 0.000,B 0.000,C 90.000,E1 33.658} C_DIS
LIN {X 0.016,Y -186.848,Z 1854.169,A 0.000,B 0.000,C 90.000,E1 30.384} C_DIS
LIN {X 0.015,Y -180.326,Z 1854.150,A 0.000,B 0.000,C 90.000,E1 27.052} C_DIS
LIN {X 0.028,Y -175.906,Z 1854.136,A 0.000,B 0.000,C 90.000,E1 24.515} C_DIS
LIN {X 0.027,Y -170.766,Z 1854.117,A 0.000,B 0.000,C 90.000,E1 21.099} C_DIS
LIN {X -0.037,Y -168.226,Z 1854.107,A 0.000,B 0.000,C 90.000,E1 19.214} C_DIS
LIN {X -0.056,Y -168.284,Z 1854.107,A 0.000,B 0.000,C 90.000,E1 19.214} C_DIS
LIN {X -0.077,Y -177.976,Z 1854.103,A 0.000,B 0.000,C 90.000,E1 18.544} C_DIS
LIN {X -0.033,Y -180.192,Z 1854.101,A 0.000,B 0.000,C 90.000,E1 18.109} C_DIS
LIN {X -0.082,Y -181.708,Z 1854.096,A 0.000,B 0.000,C 90.000,E1 17.275} C_DIS
LIN {X 0.061,Y -182.489,Z 1854.091,A 0.000,B 0.000,C 90.000,E1 16.386} C_DIS
LIN {X 0.022,Y -183.244,Z 1854.082,A 0.000,B 0.000,C 90.000,E1 14.717} C_DIS
LIN {X 0.070,Y -183.679,Z 1854.068,A 0.000,B 0.000,C 90.000,E1 12.187} C_DIS
LIN {X -0.004,Y -183.835,Z 1854.049,A 0.000,B 0.000,C 90.000,E1 8.859} C_DIS
LIN {X 0.088,Y -184.006,Z 1854.026,A 0.000,B 0.000,C 90.000,E1 4.645} C_DIS
LIN {X -0.089,Y -184.533,Z 1854.003,A 0.000,B 0.000,C 90.000,E1 0.516} C_DIS
LIN {X -0.088,Y -185.390,Z 1853.979,A 0.000,B 0.000,C 90.000,E1 356.216} C_DIS
LIN {X -0.072,Y -186.266,Z 1853.960,A 0.000,B 0.000,C 90.000,E1 352.875} C_DIS
LIN {X -0.032,Y -187.541,Z 1853.937,A 0.000,B 0.000,C 90.000,E1 348.701} C_DIS
LIN {X 0.063,Y -188.725,Z 1853.919,A 0.000,B 0.000,C 90.000,E1 345.353} C_DIS
LIN {X 0.045,Y -190.316,Z 1853.896,A 0.000,B 0.000,C 90.000,E1 341.221} C_DIS
LIN {X -0.058,Y -193.036,Z 1853.864,A 0.000,B 0.000,C 90.000,E1 335.485} C_DIS
LIN {X 0.056,Y -196.343,Z 1853.836,A 0.000,B 0.000,C 90.000,E1 330.539} C_DIS
LIN {X 0.024,Y -200.264,Z 1853.809,A 0.000,B 0.000,C 90.000,E1 325.674} C_DIS
LIN {X -0.035,Y -204.075,Z 1853.787,A 0.000,B 0.000,C 90.000,E1 321.662} C_DIS
LIN {X 0.090,Y -208.691,Z 1853.765,A 0.000,B 0.000,C 90.000,E1 317.634} C_DIS
LIN {X -0.006,Y -212.257,Z 1853.752,A 0.000,B 0.000,C 90.000,E1 315.283} C_DIS
LIN {X 0.014,Y -215.198,Z 1853.743,A 0.000,B 0.000,C 90.000,E1 313.704} C_DIS
LIN {X -0.018,Y -219.803,Z 1853.732,A 0.000,B 0.000,C 90.000,E1 311.757} C_DIS
LIN {X -0.118,Y -223.202,Z 1853.725,A 0.000,B 0.000,C 90.000,E1 310.620} C_DIS
LIN {X -0.009,Y -227.083,Z 1853.719,A 0.000,B 0.000,C 90.000,E1 309.439} C_DIS
LIN {X 0.091,Y -233.093,Z 1853.711,A 0.000,B 0.000,C 90.000,E1 307.890} C_DIS
LIN {X 0.097,Y -241.521,Z 1853.700,A 0.000,B 0.000,C 90.000,E1 306.011} C_DIS
LIN {X -0.048,Y -252.720,Z 1853.688,A 0.000,B 0.000,C 90.000,E1 303.833} C_DIS
LIN {X 0.057,Y -262.964,Z 1853.678,A 0.000,B 0.000,C 90.000,E1 302.005} C_DIS
LIN {X 0.002,Y -281.061,Z 1853.662,A 0.000,B 0.000,C 90.000,E1 299.205} C_DIS
LIN {X -0.090,Y -292.902,Z 1853.653,A 0.000,B 0.000,C 90.000,E1 297.513} C_DIS
LIN {X 0.159,Y -306.989,Z 1853.642,A 0.000,B 0.000,C 90.000,E1 295.463} C_DIS
LIN {X -0.067,Y -318.673,Z 1853.633,A 0.000,B 0.000,C 90.000,E1 293.875} C_DIS
LIN {X -0.087,Y -330.278,Z 1853.624,A 0.000,B 0.000,C 90.000,E1 292.280} C_DIS
LIN {X -0.087,Y -339.249,Z 1853.617,A 0.000,B 0.000,C 90.000,E1 291.025} C_DIS
LIN {X 0.101,Y -347.697,Z 1853.610,A 0.000,B 0.000,C 90.000,E1 289.758} C_DIS
LIN {X 0.048,Y -353.551,Z 1853.605,A 0.000,B 0.000,C 90.000,E1 288.852} C_DIS
LIN {X 0.043,Y -358.939,Z 1853.600,A 0.000,B 0.000,C 90.000,E1 287.946} C_DIS
LIN {X 0.035,Y -362.156,Z 1853.596,A 0.000,B 0.000,C 90.000,E1 287.347} C_DIS
LIN {X 0.116,Y -366.230,Z 1853.591,A 0.000,B 0.000,C 90.000,E1 286.441} C_DIS
LIN {X 0.128,Y -369.635,Z 1853.587,A 0.000,B 0.000,C 90.000,E1 285.552} C_DIS
LIN {X -0.170,Y -371.512,Z 1853.583,A 0.000,B 0.000,C 90.000,E1 285.009} C_DIS
LIN {X -0.107,Y -373.021,Z 1853.580,A 0.000,B 0.000,C 90.000,E1 284.411} C_DIS
LIN {X -0.124,Y -374.186,Z 1853.577,A 0.000,B 0.000,C 90.000,E1 283.828} C_DIS
LIN {X -0.129,Y -374.961,Z 1853.573,A 0.000,B 0.000,C 90.000,E1 283.244} C_DIS
LIN {X -0.041,Y -375.348,Z 1853.570,A 0.000,B 0.000,C 90.000,E1 282.647} C_DIS
LIN {X -0.033,Y -375.260,Z 1853.567,A 0.000,B 0.000,C 90.000,E1 282.063} C_DIS
LIN {X -0.021,Y -374.728,Z 1853.564,A 0.000,B 0.000,C 90.000,E1 281.478} C_DIS
LIN {X -0.010,Y -373.729,Z 1853.561,A 0.000,B 0.000,C 90.000,E1 280.894} C_DIS
LIN {X -0.002,Y -372.275,Z 1853.557,A 0.000,B 0.000,C 90.000,E1 280.310} C_DIS
LIN {X -0.003,Y -370.395,Z 1853.554,A 0.000,B 0.000,C 90.000,E1 279.726} C_DIS
LIN {X -0.188,Y -363.663,Z 1853.544,A 0.000,B 0.000,C 90.000,E1 277.992} C_DIS
LIN {X 0.031,Y -359.947,Z 1853.539,A 0.000,B 0.000,C 90.000,E1 277.068} C_DIS
LIN {X -0.053,Y -357.085,Z 1853.536,A 0.000,B 0.000,C 90.000,E1 276.486} C_DIS
LIN {X 0.157,Y -353.589,Z 1853.533,A 0.000,B 0.000,C 90.000,E1 275.853} C_DIS
LIN {X -0.003,Y -349.448,Z 1853.529,A 0.000,B 0.000,C 90.000,E1 275.277} C_DIS
LIN {X 0.162,Y -344.638,Z 1853.526,A 0.000,B 0.000,C 90.000,E1 274.645} C_DIS
LIN {X -0.029,Y -339.146,Z 1853.523,A 0.000,B 0.000,C 90.000,E1 274.073} C_DIS
LIN {X -0.028,Y -333.268,Z 1853.519,A 0.000,B 0.000,C 90.000,E1 273.498} C_DIS
LIN {X -0.100,Y -327.138,Z 1853.516,A 0.000,B 0.000,C 90.000,E1 272.980} C_DIS
LIN {X 0.082,Y -320.794,Z 1853.514,A 0.000,B 0.000,C 90.000,E1 272.465} C_DIS
LIN {X -0.073,Y -314.202,Z 1853.511,A 0.000,B 0.000,C 90.000,E1 272.064} C_DIS
LIN {X 0.023,Y -307.460,Z 1853.509,A 0.000,B 0.000,C 90.000,E1 271.661} C_DIS
LIN {X 0.095,Y -300.008,Z 1853.507,A 0.000,B 0.000,C 90.000,E1 271.318} C_DIS
LIN {X -0.091,Y -292.435,Z 1853.506,A 0.000,B 0.000,C 90.000,E1 271.088} C_DIS
LIN {X 0.002,Y -284.545,Z 1853.505,A 0.000,B 0.000,C 90.000,E1 270.859} C_DIS
LIN {X -0.122,Y -269.255,Z 1853.503,A 0.000,B 0.000,C 90.000,E1 270.573} C_DIS
LIN {X 0.122,Y -247.990,Z 1853.501,A 0.000,B 0.000,C 90.000,E1 270.115} C_DIS
LIN {X 0.040,Y -239.238,Z 1853.500,A 0.000,B 0.000,C 90.000,E1 270.000} C_DIS
LIN {X -0.070,Y -228.949,Z 1853.500,A 0.000,B 0.000,C 90.000,E1 269.943} C_DIS
LIN {X -0.076,Y -181.546,Z 1853.500,A 0.000,B 0.000,C 90.000,E1 269.943} C_DIS
LIN {X 0.022,Y -180.800,Z 1853.471,A 0.000,B 0.000,C 90.000,E1 264.780} C_DIS
LIN {X -0.080,Y -178.900,Z 1853.443,A 0.000,B 0.000,C 90.000,E1 259.746} C_DIS
LIN {X 0.001,Y -175.943,Z 1853.415,A 0.000,B 0.000,C 90.000,E1 254.629} C_DIS
LIN {X -0.052,Y -175.402,Z 1853.410,A 0.000,B 0.000,C 90.000,E1 253.795} C_DIS
LIN {X -0.048,Y -172.168,Z 1853.386,A 0.000,B 0.000,C 90.000,E1 249.518} C_DIS
LIN {X -0.009,Y -171.638,Z 1853.381,A 0.000,B 0.000,C 90.000,E1 248.646} C_DIS
LIN {X -0.015,Y -167.861,Z 1853.357,A 0.000,B 0.000,C 90.000,E1 244.332} C_DIS
LIN {X -0.071,Y -166.594,Z 1853.348,A 0.000,B 0.000,C 90.000,E1 242.615} C_DIS
LIN {X 0.062,Y -162.584,Z 1853.323,A 0.000,B 0.000,C 90.000,E1 238.201} C_DIS
LIN {X -0.102,Y -161.266,Z 1853.314,A 0.000,B 0.000,C 90.000,E1 236.501} C_DIS
LIN {X 0.031,Y -157.267,Z 1853.289,A 0.000,B 0.000,C 90.000,E1 232.029} C_DIS
LIN {X -0.042,Y -155.987,Z 1853.279,A 0.000,B 0.000,C 90.000,E1 230.275} C_DIS
LIN {X -0.082,Y -152.244,Z 1853.254,A 0.000,B 0.000,C 90.000,E1 225.810} C_DIS
LIN {X -0.059,Y -150.484,Z 1853.239,A 0.000,B 0.000,C 90.000,E1 223.095} C_DIS
LIN {X -0.028,Y -147.209,Z 1853.214,A 0.000,B 0.000,C 90.000,E1 218.543} C_DIS
LIN {X -0.058,Y -145.229,Z 1853.194,A 0.000,B 0.000,C 90.000,E1 214.898} C_DIS
LIN {X 0.053,Y -142.354,Z 1853.163,A 0.000,B 0.000,C 90.000,E1 209.333} C_DIS
LIN {X -0.020,Y -141.741,Z 1853.153,A 0.000,B 0.000,C 90.000,E1 207.513} C_DIS
LIN {X 0.087,Y -139.488,Z 1853.117,A 0.000,B 0.000,C 90.000,E1 200.972} C_DIS
LIN {X -0.057,Y -138.991,Z 1853.101,A 0.000,B 0.000,C 90.000,E1 198.236} C_DIS
LIN {X 0.036,Y -138.336,Z 1853.054,A 0.000,B 0.000,C 90.000,E1 189.792} C_DIS
LIN {X 0.061,Y -139.419,Z 1853.008,A 0.000,B 0.000,C 90.000,E1 181.375} C_DIS
LIN {X -0.025,Y -141.337,Z 1852.972,A 0.000,B 0.000,C 90.000,E1 174.894} C_DIS
LIN {X -0.068,Y -142.694,Z 1852.956,A 0.000,B 0.000,C 90.000,E1 172.129} C_DIS
LIN {X 0.052,Y -145.058,Z 1852.930,A 0.000,B 0.000,C 90.000,E1 167.465} C_DIS
LIN {X 0.049,Y -147.683,Z 1852.910,A 0.000,B 0.000,C 90.000,E1 163.795} C_DIS
LIN {X -0.059,Y -150.330,Z 1852.890,A 0.000,B 0.000,C 90.000,E1 160.188} C_DIS
LIN {X 0.013,Y -153.747,Z 1852.870,A 0.000,B 0.000,C 90.000,E1 156.538} C_DIS
LIN {X 0.004,Y -157.160,Z 1852.850,A 0.000,B 0.000,C 90.000,E1 152.948} C_DIS
LIN {X -0.062,Y -161.313,Z 1852.830,A 0.000,B 0.000,C 90.000,E1 149.410} C_DIS
LIN {X -0.045,Y -164.427,Z 1852.815,A 0.000,B 0.000,C 90.000,E1 146.755} C_DIS
LIN {X -0.050,Y -169.112,Z 1852.796,A 0.000,B 0.000,C 90.000,E1 143.256} C_DIS
LIN {X -0.099,Y -171.667,Z 1852.786,A 0.000,B 0.000,C 90.000,E1 141.537} C_DIS
LIN {X -0.054,Y -176.633,Z 1852.767,A 0.000,B 0.000,C 90.000,E1 138.081} C_DIS
LIN {X 0.074,Y -180.930,Z 1852.753,A 0.000,B 0.000,C 90.000,E1 135.486} C_DIS
LIN {X -0.062,Y -186.350,Z 1852.734,A 0.000,B 0.000,C 90.000,E1 132.162} C_DIS
LIN {X 0.003,Y -190.982,Z 1852.720,A 0.000,B 0.000,C 90.000,E1 129.644} C_DIS
LIN {X -0.078,Y -196.757,Z 1852.702,A 0.000,B 0.000,C 90.000,E1 126.377} C_DIS
LIN {X -0.048,Y -200.006,Z 1852.693,A 0.000,B 0.000,C 90.000,E1 124.739} C_DIS
LIN {X -0.066,Y -207.508,Z 1852.671,A 0.000,B 0.000,C 90.000,E1 120.718} C_DIS
LIN {X 0.117,Y -210.726,Z 1852.662,A 0.000,B 0.000,C 90.000,E1 119.077} C_DIS
LIN {X -0.068,Y -216.560,Z 1852.644,A 0.000,B 0.000,C 90.000,E1 115.976} C_DIS
LIN {X 0.038,Y -219.656,Z 1852.635,A 0.000,B 0.000,C 90.000,E1 114.387} C_DIS
LIN {X 0.081,Y -224.072,Z 1852.621,A 0.000,B 0.000,C 90.000,E1 111.844} C_DIS
LIN {X 0.071,Y -283.522,Z 1852.621,A 0.000,B 0.000,C 90.000,E1 111.844} C_DIS
LIN {X -0.086,Y -285.346,Z 1852.621,A 0.000,B 0.000,C 90.000,E1 111.844} C_DIS
LIN {X -0.116,Y -290.334,Z 1852.620,A 0.000,B 0.000,C 90.000,E1 111.589} C_DIS
LIN {X 0.126,Y -293.021,Z 1852.618,A 0.000,B 0.000,C 90.000,E1 111.280} C_DIS
LIN {X 0.055,Y -296.762,Z 1852.615,A 0.000,B 0.000,C 90.000,E1 110.737} C_DIS
LIN {X 0.060,Y -310.049,Z 1852.602,A 0.000,B 0.000,C 90.000,E1 108.417} C_DIS
LIN {X 0.083,Y -324.701,Z 1852.590,A 0.000,B 0.000,C 90.000,E1 106.150} C_DIS
LIN {X -0.169,Y -338.444,Z 1852.579,A 0.000,B 0.000,C 90.000,E1 104.300} C_DIS
LIN {X 0.075,Y -353.379,Z 1852.569,A 0.000,B 0.000,C 90.000,E1 102.411} C_DIS
LIN {X 0.166,Y -371.783,Z 1852.558,A 0.000,B 0.000,C 90.000,E1 100.366} C_DIS
LIN {X -0.170,Y -390.665,Z 1852.547,A 0.000,B 0.000,C 90.000,E1 98.568} C_DIS
LIN {X 0.203,Y -409.888,Z 1852.538,A 0.000,B 0.000,C 90.000,E1 96.834} C_DIS
LIN {X 0.087,Y -432.276,Z 1852.528,A 0.000,B 0.000,C 90.000,E1 95.106} C_DIS
LIN {X 0.052,Y -437.932,Z 1852.526,A 0.000,B 0.000,C 90.000,E1 94.702} C_DIS
LIN {X -0.183,Y -440.481,Z 1852.525,A 0.000,B 0.000,C 90.000,E1 94.531} C_DIS
LIN {X 0.000,Y -444.098,Z 1852.523,A 0.000,B 0.000,C 90.000,E1 94.073} C_DIS
LIN {X 0.201,Y -445.587,Z 1852.521,A 0.000,B 0.000,C 90.000,E1 93.784} C_DIS
LIN {X -0.073,Y -446.707,Z 1852.520,A 0.000,B 0.000,C 90.000,E1 93.555} C_DIS
LIN {X -0.121,Y -448.059,Z 1852.517,A 0.000,B 0.000,C 90.000,E1 93.037} C_DIS
LIN {X -0.185,Y -448.426,Z 1852.514,A 0.000,B 0.000,C 90.000,E1 92.522} C_DIS
LIN {X 0.210,Y -447.867,Z 1852.511,A 0.000,B 0.000,C 90.000,E1 91.949} C_DIS
LIN {X 0.172,Y -446.300,Z 1852.508,A 0.000,B 0.000,C 90.000,E1 91.432} C_DIS
LIN {X -0.077,Y -445.057,Z 1852.507,A 0.000,B 0.000,C 90.000,E1 91.203} C_DIS
LIN {X -0.140,Y -433.580,Z 1852.496,A 0.000,B 0.000,C 90.000,E1 89.370} C_DIS
LIN {X -0.122,Y -423.588,Z 1852.488,A 0.000,B 0.000,C 90.000,E1 87.764} C_DIS
LIN {X -0.163,Y -411.804,Z 1852.477,A 0.000,B 0.000,C 90.000,E1 85.869} C_DIS
LIN {X -0.002,Y -399.926,Z 1852.466,A 0.000,B 0.000,C 90.000,E1 83.913} C_DIS
LIN {X -0.058,Y -387.973,Z 1852.455,A 0.000,B 0.000,C 90.000,E1 81.951} C_DIS
LIN {X 0.068,Y -376.058,Z 1852.444,A 0.000,B 0.000,C 90.000,E1 79.926} C_DIS
LIN {X 0.067,Y -359.471,Z 1852.428,A 0.000,B 0.000,C 90.000,E1 76.992} C_DIS
LIN {X 0.097,Y -343.938,Z 1852.411,A 0.000,B 0.000,C 90.000,E1 73.976} C_DIS
LIN {X 0.096,Y -331.991,Z 1852.397,A 0.000,B 0.000,C 90.000,E1 71.511} C_DIS
LIN {X -0.091,Y -320.297,Z 1852.383,A 0.000,B 0.000,C 90.000,E1 69.028} C_DIS
LIN {X 0.106,Y -307.720,Z 1852.367,A 0.000,B 0.000,C 90.000,E1 66.102} C_DIS
LIN {X 0.050,Y -298.150,Z 1852.355,A 0.000,B 0.000,C 90.000,E1 63.819} C_DIS
LIN {X -0.096,Y -287.434,Z 1852.340,A 0.000,B 0.000,C 90.000,E1 61.179} C_DIS
LIN {X -0.047,Y -278.029,Z 1852.327,A 0.000,B 0.000,C 90.000,E1 58.791} C_DIS
LIN {X -0.061,Y -268.576,Z 1852.313,A 0.000,B 0.000,C 90.000,E1 56.373} C_DIS
LIN {X -0.116,Y -260.391,Z 1852.301,A 0.000,B 0.000,C 90.000,E1 54.276} C_DIS
LIN {X 0.010,Y -250.786,Z 1852.287,A 0.000,B 0.000,C 90.000,E1 51.743} C_DIS
LIN {X 0.079,Y -241.245,Z 1852.273,A 0.000,B 0.000,C 90.000,E1 49.175} C_DIS
LIN {X 0.004,Y -230.547,Z 1852.257,A 0.000,B 0.000,C 90.000,E1 46.215} C_DIS
LIN {X -0.007,Y -220.360,Z 1852.240,A 0.000,B 0.000,C 90.000,E1 43.176} C_DIS
LIN {X -0.093,Y -210.740,Z 1852.223,A 0.000,B 0.000,C 90.000,E1 40.092} C_DIS
LIN {X 0.098,Y -201.978,Z 1852.205,A 0.000,B 0.000,C 90.000,E1 36.870} C_DIS
LIN {X 0.055,Y -194.053,Z 1852.187,A 0.000,B 0.000,C 90.000,E1 33.658} C_DIS
LIN {X 0.035,Y -186.852,Z 1852.169,A 0.000,B 0.000,C 90.000,E1 30.384} C_DIS
LIN {X 0.033,Y -180.330,Z 1852.150,A 0.000,B 0.000,C 90.000,E1 27.052} C_DIS
LIN {X 0.047,Y -175.909,Z 1852.136,A 0.000,B 0.000,C 90.000,E1 24.515} C_DIS
LIN {X 0.014,Y -172.626,Z 1852.125,A 0.000,B 0.000,C 90.000,E1 22.408} C_DIS
LIN {X 0.060,Y -172.694,Z 1852.125,A 0.000,B 0.000,C 90.000,E1 22.386} C_DIS
LIN {X -0.038,Y -180.875,Z 1852.121,A 0.000,B 0.000,C 90.000,E1 21.716} C_DIS
LIN {X 0.093,Y -183.057,Z 1852.119,A 0.000,B 0.000,C 90.000,E1 21.408} C_DIS
LIN {X -0.101,Y -184.771,Z 1852.115,A 0.000,B 0.000,C 90.000,E1 20.737} C_DIS
LIN {X -0.058,Y -185.608,Z 1852.110,A 0.000,B 0.000,C 90.000,E1 19.885} C_DIS
LIN {X -0.005,Y -186.042,Z 1852.106,A 0.000,B 0.000,C 90.000,E1 19.033} C_DIS
LIN {X 0.056,Y -186.422,Z 1852.096,A 0.000,B 0.000,C 90.000,E1 17.347} C_DIS
LIN {X -0.053,Y -186.378,Z 1852.083,A 0.000,B 0.000,C 90.000,E1 14.883} C_DIS
LIN {X 0.007,Y -185.953,Z 1852.064,A 0.000,B 0.000,C 90.000,E1 11.535} C_DIS
LIN {X 0.054,Y -185.426,Z 1852.041,A 0.000,B 0.000,C 90.000,E1 7.352} C_DIS
LIN {X 0.041,Y -185.289,Z 1852.013,A 0.000,B 0.000,C 90.000,E1 2.350} C_DIS
LIN {X -0.052,Y -185.691,Z 1851.988,A 0.000,B 0.000,C 90.000,E1 357.879} C_DIS
LIN {X 0.033,Y -186.430,Z 1851.965,A 0.000,B 0.000,C 90.000,E1 353.685} C_DIS
LIN {X 0.080,Y -187.399,Z 1851.942,A 0.000,B 0.000,C 90.000,E1 349.511} C_DIS
LIN {X -0.078,Y -188.601,Z 1851.919,A 0.000,B 0.000,C 90.000,E1 345.408} C_DIS
LIN {X 0.082,Y -189.988,Z 1851.896,A 0.000,B 0.000,C 90.000,E1 341.221} C_DIS
LIN {X -0.034,Y -192.733,Z 1851.864,A 0.000,B 0.000,C 90.000,E1 335.485} C_DIS
LIN {X 0.070,Y -196.087,Z 1851.836,A 0.000,B 0.000,C 90.000,E1 330.539} C_DIS
LIN {X 0.029,Y -200.019,Z 1851.809,A 0.000,B 0.000,C 90.000,E1 325.674} C_DIS
LIN {X -0.038,Y -203.881,Z 1851.787,A 0.000,B 0.000,C 90.000,E1 321.662} C_DIS
LIN {X 0.082,Y -208.566,Z 1851.765,A 0.000,B 0.000,C 90.000,E1 317.634} C_DIS
LIN {X -0.017,Y -212.160,Z 1851.752,A 0.000,B 0.000,C 90.000,E1 315.283} C_DIS
LIN {X 0.001,Y -215.163,Z 1851.743,A 0.000,B 0.000,C 90.000,E1 313.704} C_DIS
LIN {X -0.031,Y -219.804,Z 1851.732,A 0.000,B 0.000,C 90.000,E1 311.757} C_DIS
LIN {X -0.132,Y -223.245,Z 1851.725,A 0.000,B 0.000,C 90.000,E1 310.620} C_DIS
LIN {X -0.022,Y -227.165,Z 1851.719,A 0.000,B 0.000,C 90.000,E1 309.439} C_DIS
LIN {X 0.079,Y -233.214,Z 1851.711,A 0.000,B 0.000,C 90.000,E1 307.890} C_DIS
LIN {X 0.086,Y -241.700,Z 1851.700,A 0.000,B 0.000,C 90.000,E1 306.011} C_DIS
LIN {X -0.056,Y -252.925,Z 1851.688,A 0.000,B 0.000,C 90.000,E1 303.833} C_DIS
LIN {X 0.052,Y -263.204,Z 1851.678,A 0.000,B 0.000,C 90.000,E1 302.005} C_DIS
LIN {X 0.003,Y -281.352,Z 1851.662,A 0.000,B 0.000,C 90.000,E1 299.205} C_DIS
LIN {X -0.084,Y -293.219,Z 1851.653,A 0.000,B 0.000,C 90.000,E1 297.513} C_DIS
LIN {X 0.172,Y -307.377,Z 1851.642,A 0.000,B 0.000,C 90.000,E1 295.463} C_DIS
LIN {X -0.177,Y -319.086,Z 1851.633,A 0.000,B 0.000,C 90.000,E1 293.898} C_DIS
LIN {X -0.059,Y -330.774,Z 1851.624,A 0.000,B 0.000,C 90.000,E1 292.280} C_DIS
LIN {X -0.174,Y -339.767,Z 1851.617,A 0.000,B 0.000,C 90.000,E1 291.046} C_DIS
LIN {X 0.137,Y -346.188,Z 1851.612,A 0.000,B 0.000,C 90.000,E1 290.066} C_DIS
LIN {X 0.180,Y -352.259,Z 1851.606,A 0.000,B 0.000,C 90.000,E1 289.141} C_DIS
LIN {X 0.098,Y -359.558,Z 1851.600,A 0.000,B 0.000,C 90.000,E1 287.946} C_DIS
LIN {X 0.093,Y -362.747,Z 1851.596,A 0.000,B 0.000,C 90.000,E1 287.347} C_DIS
LIN {X 0.111,Y -365.568,Z 1851.593,A 0.000,B 0.000,C 90.000,E1 286.749} C_DIS
LIN {X -0.132,Y -369.160,Z 1851.588,A 0.000,B 0.000,C 90.000,E1 285.898} C_DIS
LIN {X -0.095,Y -372.095,Z 1851.583,A 0.000,B 0.000,C 90.000,E1 285.009} C_DIS
LIN {X -0.028,Y -373.612,Z 1851.580,A 0.000,B 0.000,C 90.000,E1 284.411} C_DIS
LIN {X -0.041,Y -374.751,Z 1851.577,A 0.000,B 0.000,C 90.000,E1 283.828} C_DIS
LIN {X -0.042,Y -375.496,Z 1851.573,A 0.000,B 0.000,C 90.000,E1 283.244} C_DIS
LIN {X 0.049,Y -375.847,Z 1851.570,A 0.000,B 0.000,C 90.000,E1 282.647} C_DIS
LIN {X 0.060,Y -375.748,Z 1851.567,A 0.000,B 0.000,C 90.000,E1 282.063} C_DIS
LIN {X 0.075,Y -375.226,Z 1851.564,A 0.000,B 0.000,C 90.000,E1 281.478} C_DIS
LIN {X 0.088,Y -374.173,Z 1851.561,A 0.000,B 0.000,C 90.000,E1 280.894} C_DIS
LIN {X 0.098,Y -372.668,Z 1851.557,A 0.000,B 0.000,C 90.000,E1 280.310} C_DIS
LIN {X 0.036,Y -369.671,Z 1851.552,A 0.000,B 0.000,C 90.000,E1 279.443} C_DIS
LIN {X -0.143,Y -361.598,Z 1851.541,A 0.000,B 0.000,C 90.000,E1 277.409} C_DIS
LIN {X 0.097,Y -358.891,Z 1851.538,A 0.000,B 0.000,C 90.000,E1 276.777} C_DIS
LIN {X -0.034,Y -355.744,Z 1851.534,A 0.000,B 0.000,C 90.000,E1 276.201} C_DIS
LIN {X -0.180,Y -351.978,Z 1851.531,A 0.000,B 0.000,C 90.000,E1 275.625} C_DIS
LIN {X 0.004,Y -347.496,Z 1851.528,A 0.000,B 0.000,C 90.000,E1 274.992} C_DIS
LIN {X 0.158,Y -342.287,Z 1851.524,A 0.000,B 0.000,C 90.000,E1 274.359} C_DIS
LIN {X 0.040,Y -336.548,Z 1851.521,A 0.000,B 0.000,C 90.000,E1 273.784} C_DIS
LIN {X 0.153,Y -330.529,Z 1851.518,A 0.000,B 0.000,C 90.000,E1 273.212} C_DIS
LIN {X -0.125,Y -324.261,Z 1851.515,A 0.000,B 0.000,C 90.000,E1 272.751} C_DIS
LIN {X -0.115,Y -317.821,Z 1851.513,A 0.000,B 0.000,C 90.000,E1 272.293} C_DIS
LIN {X -0.158,Y -311.162,Z 1851.510,A 0.000,B 0.000,C 90.000,E1 271.892} C_DIS
LIN {X 0.028,Y -303.803,Z 1851.508,A 0.000,B 0.000,C 90.000,E1 271.489} C_DIS
LIN {X 0.011,Y -296.625,Z 1851.507,A 0.000,B 0.000,C 90.000,E1 271.203} C_DIS
LIN {X -0.054,Y -288.561,Z 1851.505,A 0.000,B 0.000,C 90.000,E1 270.974} C_DIS
LIN {X -0.094,Y -281.066,Z 1851.504,A 0.000,B 0.000,C 90.000,E1 270.802} C_DIS
LIN {X -0.057,Y -251.989,Z 1851.501,A 0.000,B 0.000,C 90.000,E1 270.229} C_DIS
LIN {X 0.086,Y -243.852,Z 1851.500,A 0.000,B 0.000,C 90.000,E1 270.057} C_DIS
LIN {X -0.080,Y -236.345,Z 1851.500,A 0.000,B 0.000,C 90.000,E1 270.000} C_DIS
LIN {X -0.048,Y -227.826,Z 1851.500,A 0.000,B 0.000,C 90.000,E1 269.943} C_DIS
LIN {X -0.057,Y -181.547,Z 1851.500,A 0.000,B 0.000,C 90.000,E1 269.943} C_DIS
LIN {X 0.063,Y -180.804,Z 1851.471,A 0.000,B 0.000,C 90.000,E1 264.780} C_DIS
LIN {X -0.041,Y -178.905,Z 1851.443,A 0.000,B 0.000,C 90.000,E1 259.746} C_DIS
LIN {X 0.040,Y -175.949,Z 1851.415,A 0.000,B 0.000,C 90.000,E1 254.629} C_DIS
LIN {X -0.013,Y -175.412,Z 1851.410,A 0.000,B 0.000,C 90.000,E1 253.795} C_DIS
LIN {X -0.010,Y -172.176,Z 1851.386,A 0.000,B 0.000,C 90.000,E1 249.518} C_DIS
LIN {X 0.029,Y -171.647,Z 1851.381,A 0.000,B 0.000,C 90.000,E1 248.646} C_DIS
LIN {X 0.024,Y -167.870,Z 1851.357,A 0.000,B 0.000,C 90.000,E1 244.332} C_DIS
LIN {X -0.033,Y -166.605,Z 1851.348,A 0.000,B 0.000,C 90.000,E1 242.615} C_DIS
LIN {X -0.039,Y -162.594,Z 1851.323,A 0.000,B 0.000,C 90.000,E1 238.250} C_DIS
LIN {X -0.065,Y -161.278,Z 1851.314,A 0.000,B 0.000,C 90.000,E1 236.501} C_DIS
LIN {X -0.030,Y -157.277,Z 1851.289,A 0.000,B 0.000,C 90.000,E1 232.065} C_DIS
LIN {X -0.006,Y -155.996,Z 1851.279,A 0.000,B 0.000,C 90.000,E1 230.275} C_DIS
LIN {X -0.046,Y -152.253,Z 1851.254,A 0.000,B 0.000,C 90.000,E1 225.810} C_DIS
LIN {X -0.023,Y -150.493,Z 1851.239,A 0.000,B 0.000,C 90.000,E1 223.095} C_DIS
LIN {X 0.007,Y -147.216,Z 1851.214,A 0.000,B 0.000,C 90.000,E1 218.543} C_DIS
LIN {X -0.024,Y -145.238,Z 1851.194,A 0.000,B 0.000,C 90.000,E1 214.898} C_DIS
LIN {X 0.017,Y -142.360,Z 1851.163,A 0.000,B 0.000,C 90.000,E1 209.361} C_DIS
LIN {X 0.014,Y -141.746,Z 1851.153,A 0.000,B 0.000,C 90.000,E1 207.513} C_DIS
LIN {X -0.059,Y -139.491,Z 1851.117,A 0.000,B 0.000,C 90.000,E1 201.046} C_DIS
LIN {X -0.022,Y -138.995,Z 1851.101,A 0.000,B 0.000,C 90.000,E1 198.236} C_DIS
LIN {X -0.066,Y -138.336,Z 1851.055,A 0.000,B 0.000,C 90.000,E1 189.849} C_DIS
LIN {X -0.044,Y -139.415,Z 1851.008,A 0.000,B 0.000,C 90.000,E1 181.432} C_DIS
LIN {X 0.009,Y -141.331,Z 1850.972,A 0.000,B 0.000,C 90.000,E1 174.894} C_DIS
LIN {X -0.033,Y -142.688,Z 1850.956,A 0.000,B 0.000,C 90.000,E1 172.129} C_DIS
LIN {X -0.055,Y -145.050,Z 1850.931,A 0.000,B 0.000,C 90.000,E1 167.521} C_DIS
LIN {X 0.084,Y -147.675,Z 1850.910,A 0.000,B 0.000,C 90.000,E1 163.795} C_DIS
LIN {X -0.023,Y -150.318,Z 1850.890,A 0.000,B 0.000,C 90.000,E1 160.188} C_DIS
LIN {X 0.049,Y -153.732,Z 1850.870,A 0.000,B 0.000,C 90.000,E1 156.538} C_DIS
LIN {X 0.040,Y -157.146,Z 1850.850,A 0.000,B 0.000,C 90.000,E1 152.948} C_DIS
LIN {X -0.025,Y -161.295,Z 1850.830,A 0.000,B 0.000,C 90.000,E1 149.410} C_DIS
LIN {X -0.008,Y -164.412,Z 1850.815,A 0.000,B 0.000,C 90.000,E1 146.755} C_DIS
LIN {X -0.011,Y -169.093,Z 1850.796,A 0.000,B 0.000,C 90.000,E1 143.256} C_DIS
LIN {X -0.060,Y -171.650,Z 1850.786,A 0.000,B 0.000,C 90.000,E1 141.537} C_DIS
LIN {X -0.014,Y -176.613,Z 1850.767,A 0.000,B 0.000,C 90.000,E1 138.081} C_DIS
LIN {X -0.013,Y -180.911,Z 1850.753,A 0.000,B 0.000,C 90.000,E1 135.526} C_DIS
LIN {X -0.022,Y -186.327,Z 1850.734,A 0.000,B 0.000,C 90.000,E1 132.162} C_DIS
LIN {X 0.045,Y -190.961,Z 1850.720,A 0.000,B 0.000,C 90.000,E1 129.644} C_DIS
LIN {X -0.036,Y -196.733,Z 1850.702,A 0.000,B 0.000,C 90.000,E1 126.377} C_DIS
LIN {X -0.006,Y -199.980,Z 1850.693,A 0.000,B 0.000,C 90.000,E1 124.739} C_DIS
LIN {X -0.022,Y -207.484,Z 1850.671,A 0.000,B 0.000,C 90.000,E1 120.718} C_DIS
LIN {X -0.024,Y -210.705,Z 1850.662,A 0.000,B 0.000,C 90.000,E1 119.127} C_DIS
LIN {X -0.024,Y -216.537,Z 1850.644,A 0.000,B 0.000,C 90.000,E1 115.976} C_DIS
LIN {X 0.082,Y -219.638,Z 1850.636,A 0.000,B 0.000,C 90.000,E1 114.387} C_DIS
LIN {X 0.101,Y -224.063,Z 1850.621,A 0.000,B 0.000,C 90.000,E1 111.844} C_DIS
LIN {X 0.096,Y -282.801,Z 1850.621,A 0.000,B 0.000,C 90.000,E1 111.844} C_DIS
LIN {X -0.029,Y -284.940,Z 1850.621,A 0.000,B 0.000,C 90.000,E1 111.844} C_DIS
LIN {X -0.058,Y -290.201,Z 1850.620,A 0.000,B 0.000,C 90.000,E1 111.589} C_DIS
LIN {X -0.088,Y -292.925,Z 1850.618,A 0.000,B 0.000,C 90.000,E1 111.334} C_DIS
LIN {X -0.130,Y -296.665,Z 1850.615,A 0.000,B 0.000,C 90.000,E1 110.791} C_DIS
LIN {X 0.155,Y -309.942,Z 1850.602,A 0.000,B 0.000,C 90.000,E1 108.417} C_DIS
LIN {X -0.132,Y -324.582,Z 1850.590,A 0.000,B 0.000,C 90.000,E1 106.205} C_DIS
LIN {X -0.071,Y -338.316,Z 1850.579,A 0.000,B 0.000,C 90.000,E1 104.300} C_DIS
LIN {X 0.174,Y -353.239,Z 1850.569,A 0.000,B 0.000,C 90.000,E1 102.411} C_DIS
LIN {X -0.106,Y -371.641,Z 1850.558,A 0.000,B 0.000,C 90.000,E1 100.423} C_DIS
LIN {X -0.079,Y -390.519,Z 1850.547,A 0.000,B 0.000,C 90.000,E1 98.568} C_DIS
LIN {X -0.117,Y -409.740,Z 1850.538,A 0.000,B 0.000,C 90.000,E1 96.891} C_DIS
LIN {X 0.169,Y -432.125,Z 1850.528,A 0.000,B 0.000,C 90.000,E1 95.106} C_DIS
LIN {X 0.134,Y -437.780,Z 1850.526,A 0.000,B 0.000,C 90.000,E1 94.702} C_DIS
LIN {X -0.103,Y -440.362,Z 1850.525,A 0.000,B 0.000,C 90.000,E1 94.531} C_DIS
LIN {X 0.111,Y -443.995,Z 1850.523,A 0.000,B 0.000,C 90.000,E1 94.073} C_DIS
LIN {X -0.133,Y -445.507,Z 1850.521,A 0.000,B 0.000,C 90.000,E1 93.841} C_DIS
LIN {X 0.037,Y -446.644,Z 1850.520,A 0.000,B 0.000,C 90.000,E1 93.555} C_DIS
LIN {X -0.010,Y -448.024,Z 1850.517,A 0.000,B 0.000,C 90.000,E1 93.037} C_DIS
LIN {X -0.075,Y -448.414,Z 1850.514,A 0.000,B 0.000,C 90.000,E1 92.522} C_DIS
LIN {X -0.128,Y -447.878,Z 1850.511,A 0.000,B 0.000,C 90.000,E1 92.007} C_DIS
LIN {X -0.165,Y -446.339,Z 1850.508,A 0.000,B 0.000,C 90.000,E1 91.489} C_DIS
LIN {X 0.032,Y -445.116,Z 1850.507,A 0.000,B 0.000,C 90.000,E1 91.203} C_DIS
LIN {X -0.033,Y -433.648,Z 1850.496,A 0.000,B 0.000,C 90.000,E1 89.370} C_DIS
LIN {X -0.016,Y -423.661,Z 1850.488,A 0.000,B 0.000,C 90.000,E1 87.764} C_DIS
LIN {X -0.058,Y -411.876,Z 1850.477,A 0.000,B 0.000,C 90.000,E1 85.869} C_DIS
LIN {X 0.101,Y -399.998,Z 1850.466,A 0.000,B 0.000,C 90.000,E1 83.913} C_DIS
LIN {X 0.043,Y -388.047,Z 1850.455,A 0.000,B 0.000,C 90.000,E1 81.951} C_DIS
LIN {X -0.202,Y -376.129,Z 1850.444,A 0.000,B 0.000,C 90.000,E1 79.982} C_DIS
LIN {X 0.165,Y -359.535,Z 1850.428,A 0.000,B 0.000,C 90.000,E1 76.992} C_DIS
LIN {X 0.192,Y -343.997,Z 1850.411,A 0.000,B 0.000,C 90.000,E1 73.976} C_DIS
LIN {X 0.083,Y -332.048,Z 1850.397,A 0.000,B 0.000,C 90.000,E1 71.529} C_DIS
LIN {X 0.000,Y -320.350,Z 1850.384,A 0.000,B 0.000,C 90.000,E1 69.028} C_DIS
LIN {X 0.070,Y -307.770,Z 1850.367,A 0.000,B 0.000,C 90.000,E1 66.125} C_DIS
LIN {X 0.006,Y -298.196,Z 1850.355,A 0.000,B 0.000,C 90.000,E1 63.845} C_DIS
LIN {X -0.011,Y -287.479,Z 1850.340,A 0.000,B 0.000,C 90.000,E1 61.179} C_DIS
LIN {X 0.038,Y -278.076,Z 1850.327,A 0.000,B 0.000,C 90.000,E1 58.791} C_DIS
LIN {X 0.020,Y -268.624,Z 1850.313,A 0.000,B 0.000,C 90.000,E1 56.373} C_DIS
LIN {X -0.036,Y -260.441,Z 1850.302,A 0.000,B 0.000,C 90.000,E1 54.276} C_DIS
LIN {X 0.064,Y -252.220,Z 1850.290,A 0.000,B 0.000,C 90.000,E1 52.110} C_DIS
LIN {X -0.027,Y -242.635,Z 1850.275,A 0.000,B 0.000,C 90.000,E1 49.585} C_DIS
LIN {X -0.003,Y -233.222,Z 1850.261,A 0.000,B 0.000,C 90.000,E1 46.986} C_DIS
LIN {X 0.049,Y -222.925,Z 1850.244,A 0.000,B 0.000,C 90.000,E1 43.947} C_DIS
LIN {X 0.022,Y -213.118,Z 1850.227,A 0.000,B 0.000,C 90.000,E1 40.862} C_DIS
LIN {X -0.057,Y -204.111,Z 1850.209,A 0.000,B 0.000,C 90.000,E1 37.729} C_DIS
LIN {X 0.069,Y -196.012,Z 1850.192,A 0.000,B 0.000,C 90.000,E1 34.485} C_DIS
LIN {X -0.062,Y -188.606,Z 1850.174,A 0.000,B 0.000,C 90.000,E1 31.258} C_DIS
LIN {X 0.073,Y -181.919,Z 1850.155,A 0.000,B 0.000,C 90.000,E1 27.897} C_DIS
LIN {X 0.082,Y -177.514,Z 1850.142,A 0.000,B 0.000,C 90.000,E1 25.463} C_DIS
LIN {X 0.061,Y -177.509,Z 1850.142,A 0.000,B 0.000,C 90.000,E1 25.463} C_DIS
LIN {X 0.001,Y -184.571,Z 1850.138,A 0.000,B 0.000,C 90.000,E1 24.771} C_DIS
LIN {X -0.106,Y -188.006,Z 1850.134,A 0.000,B 0.000,C 90.000,E1 24.207} C_DIS
LIN {X 0.016,Y -189.211,Z 1850.130,A 0.000,B 0.000,C 90.000,E1 23.334} C_DIS
LIN {X -0.016,Y -189.714,Z 1850.125,A 0.000,B 0.000,C 90.000,E1 22.514} C_DIS
LIN {X 0.064,Y -189.929,Z 1850.120,A 0.000,B 0.000,C 90.000,E1 21.663} C_DIS
LIN {X -0.055,Y -189.907,Z 1850.111,A 0.000,B 0.000,C 90.000,E1 20.047} C_DIS
LIN {X -0.101,Y -189.399,Z 1850.098,A 0.000,B 0.000,C 90.000,E1 17.583} C_DIS
LIN {X 0.026,Y -188.710,Z 1850.084,A 0.000,B 0.000,C 90.000,E1 15.064} C_DIS
LIN {X -0.069,Y -187.466,Z 1850.061,A 0.000,B 0.000,C 90.000,E1 10.950} C_DIS
LIN {X -0.077,Y -186.376,Z 1850.033,A 0.000,B 0.000,C 90.000,E1 5.967} C_DIS
LIN {X -0.088,Y -186.026,Z 1850.005,A 0.000,B 0.000,C 90.000,E1 0.974} C_DIS
LIN {X -0.056,Y -186.277,Z 1849.979,A 0.000,B 0.000,C 90.000,E1 356.216} C_DIS
LIN {X -0.019,Y -186.735,Z 1849.960,A 0.000,B 0.000,C 90.000,E1 352.875} C_DIS
LIN {X 0.032,Y -187.490,Z 1849.937,A 0.000,B 0.000,C 90.000,E1 348.701} C_DIS
LIN {X -0.042,Y -188.525,Z 1849.914,A 0.000,B 0.000,C 90.000,E1 344.574} C_DIS
LIN {X -0.006,Y -189.999,Z 1849.891,A 0.000,B 0.000,C 90.000,E1 340.423} C_DIS
LIN {X -0.045,Y -192.930,Z 1849.859,A 0.000,B 0.000,C 90.000,E1 334.665} C_DIS
LIN {X 0.054,Y -195.816,Z 1849.836,A 0.000,B 0.000,C 90.000,E1 330.539} C_DIS
LIN {X 0.004,Y -199.784,Z 1849.809,A 0.000,B 0.000,C 90.000,E1 325.674} C_DIS
LIN {X 0.090,Y -203.701,Z 1849.787,A 0.000,B 0.000,C 90.000,E1 321.618} C_DIS
LIN {X 0.044,Y -208.447,Z 1849.765,A 0.000,B 0.000,C 90.000,E1 317.634} C_DIS
LIN {X 0.091,Y -212.077,Z 1849.751,A 0.000,B 0.000,C 90.000,E1 315.243} C_DIS
LIN {X -0.043,Y -215.096,Z 1849.743,A 0.000,B 0.000,C 90.000,E1 313.704} C_DIS
LIN {X -0.077,Y -219.844,Z 1849.732,A 0.000,B 0.000,C 90.000,E1 311.757} C_DIS
LIN {X 0.137,Y -223.306,Z 1849.725,A 0.000,B 0.000,C 90.000,E1 310.539} C_DIS
LIN {X -0.068,Y -227.292,Z 1849.719,A 0.000,B 0.000,C 90.000,E1 309.439} C_DIS
LIN {X 0.033,Y -233.364,Z 1849.711,A 0.000,B 0.000,C 90.000,E1 307.890} C_DIS
LIN {X 0.041,Y -241.918,Z 1849.700,A 0.000,B 0.000,C 90.000,E1 306.011} C_DIS
LIN {X 0.111,Y -253.178,Z 1849.688,A 0.000,B 0.000,C 90.000,E1 303.785} C_DIS
LIN {X 0.012,Y -263.483,Z 1849.678,A 0.000,B 0.000,C 90.000,E1 302.005} C_DIS
LIN {X 0.024,Y -279.354,Z 1849.664,A 0.000,B 0.000,C 90.000,E1 299.539} C_DIS
LIN {X -0.114,Y -293.584,Z 1849.653,A 0.000,B 0.000,C 90.000,E1 297.513} C_DIS
LIN {X 0.148,Y -307.814,Z 1849.642,A 0.000,B 0.000,C 90.000,E1 295.463} C_DIS
LIN {X 0.150,Y -321.936,Z 1849.631,A 0.000,B 0.000,C 90.000,E1 293.515} C_DIS
LIN {X -0.104,Y -333.628,Z 1849.622,A 0.000,B 0.000,C 90.000,E1 291.972} C_DIS
LIN {X -0.186,Y -342.549,Z 1849.615,A 0.000,B 0.000,C 90.000,E1 290.737} C_DIS
LIN {X 0.147,Y -348.852,Z 1849.610,A 0.000,B 0.000,C 90.000,E1 289.758} C_DIS
LIN {X 0.104,Y -354.777,Z 1849.605,A 0.000,B 0.000,C 90.000,E1 288.852} C_DIS
LIN {X 0.113,Y -360.174,Z 1849.600,A 0.000,B 0.000,C 90.000,E1 287.946} C_DIS
LIN {X 0.113,Y -363.356,Z 1849.596,A 0.000,B 0.000,C 90.000,E1 287.347} C_DIS
LIN {X -0.217,Y -366.194,Z 1849.593,A 0.000,B 0.000,C 90.000,E1 286.804} C_DIS
LIN {X -0.104,Y -369.788,Z 1849.588,A 0.000,B 0.000,C 90.000,E1 285.898} C_DIS
LIN {X -0.061,Y -372.672,Z 1849.583,A 0.000,B 0.000,C 90.000,E1 285.009} C_DIS
LIN {X 0.010,Y -374.205,Z 1849.580,A 0.000,B 0.000,C 90.000,E1 284.411} C_DIS
LIN {X 0.000,Y -375.340,Z 1849.577,A 0.000,B 0.000,C 90.000,E1 283.828} C_DIS
LIN {X 0.003,Y -376.011,Z 1849.574,A 0.000,B 0.000,C 90.000,E1 283.244} C_DIS
LIN {X 0.098,Y -376.348,Z 1849.570,A 0.000,B 0.000,C 90.000,E1 282.647} C_DIS
LIN {X 0.113,Y -376.215,Z 1849.567,A 0.000,B 0.000,C 90.000,E1 282.063} C_DIS
LIN {X 0.130,Y -375.650,Z 1849.564,A 0.000,B 0.000,C 90.000,E1 281.478} C_DIS
LIN {X 0.146,Y -374.566,Z 1849.561,A 0.000,B 0.000,C 90.000,E1 280.894} C_DIS
LIN {X 0.159,Y -373.077,Z 1849.557,A 0.000,B 0.000,C 90.000,E1 280.310} C_DIS
LIN {X 0.100,Y -369.953,Z 1849.552,A 0.000,B 0.000,C 90.000,E1 279.443} C_DIS
LIN {X -0.046,Y -363.037,Z 1849.543,A 0.000,B 0.000,C 90.000,E1 277.701} C_DIS
LIN {X 0.166,Y -359.132,Z 1849.538,A 0.000,B 0.000,C 90.000,E1 276.777} C_DIS
LIN {X 0.036,Y -356.005,Z 1849.534,A 0.000,B 0.000,C 90.000,E1 276.201} C_DIS
LIN {X -0.109,Y -352.234,Z 1849.531,A 0.000,B 0.000,C 90.000,E1 275.625} C_DIS
LIN {X 0.076,Y -347.790,Z 1849.528,A 0.000,B 0.000,C 90.000,E1 274.992} C_DIS
LIN {X -0.111,Y -342.561,Z 1849.524,A 0.000,B 0.000,C 90.000,E1 274.416} C_DIS
LIN {X 0.129,Y -336.861,Z 1849.521,A 0.000,B 0.000,C 90.000,E1 273.784} C_DIS
LIN {X -0.070,Y -330.859,Z 1849.518,A 0.000,B 0.000,C 90.000,E1 273.269} C_DIS
LIN {X -0.012,Y -324.652,Z 1849.515,A 0.000,B 0.000,C 90.000,E1 272.751} C_DIS
LIN {X -0.036,Y -318.130,Z 1849.513,A 0.000,B 0.000,C 90.000,E1 272.293} C_DIS
LIN {X -0.061,Y -311.510,Z 1849.510,A 0.000,B 0.000,C 90.000,E1 271.892} C_DIS
LIN {X 0.144,Y -304.405,Z 1849.508,A 0.000,B 0.000,C 90.000,E1 271.489} C_DIS
LIN {X 0.047,Y -296.787,Z 1849.507,A 0.000,B 0.000,C 90.000,E1 271.203} C_DIS
LIN {X 0.013,Y -289.063,Z 1849.505,A 0.000,B 0.000,C 90.000,E1 270.974} C_DIS
LIN {X -0.110,Y -277.935,Z 1849.504,A 0.000,B 0.000,C 90.000,E1 270.745} C_DIS
LIN {X 0.033,Y -252.864,Z 1849.501,A 0.000,B 0.000,C 90.000,E1 270.229} C_DIS
LIN {X -0.083,Y -240.556,Z 1849.500,A 0.000,B 0.000,C 90.000,E1 270.057} C_DIS
LIN {X -0.016,Y -227.904,Z 1849.500,A 0.000,B 0.000,C 90.000,E1 269.943} C_DIS
LIN {X -0.033,Y -181.549,Z 1849.500,A 0.000,B 0.000,C 90.000,E1 269.943} C_DIS
LIN {X -0.079,Y -180.809,Z 1849.471,A 0.000,B 0.000,C 90.000,E1 264.837} C_DIS
LIN {X -0.002,Y -178.910,Z 1849.443,A 0.000,B 0.000,C 90.000,E1 259.746} C_DIS
LIN {X 0.078,Y -175.954,Z 1849.415,A 0.000,B 0.000,C 90.000,E1 254.629} C_DIS
LIN {X 0.025,Y -175.423,Z 1849.410,A 0.000,B 0.000,C 90.000,E1 253.795} C_DIS
LIN {X 0.027,Y -172.184,Z 1849.386,A 0.000,B 0.000,C 90.000,E1 249.518} C_DIS
LIN {X 0.066,Y -171.656,Z 1849.381,A 0.000,B 0.000,C 90.000,E1 248.646} C_DIS
LIN {X 0.060,Y -167.880,Z 1849.358,A 0.000,B 0.000,C 90.000,E1 244.332} C_DIS
LIN {X 0.003,Y -166.616,Z 1849.348,A 0.000,B 0.000,C 90.000,E1 242.615} C_DIS
LIN {X -0.003,Y -162.603,Z 1849.324,A 0.000,B 0.000,C 90.000,E1 238.250} C_DIS
LIN {X -0.029,Y -161.288,Z 1849.314,A 0.000,B 0.000,C 90.000,E1 236.501} C_DIS
LIN {X 0.006,Y -157.287,Z 1849.289,A 0.000,B 0.000,C 90.000,E1 232.065} C_DIS
LIN {X 0.029,Y -156.005,Z 1849.279,A 0.000,B 0.000,C 90.000,E1 230.275} C_DIS
LIN {X -0.012,Y -152.263,Z 1849.255,A 0.000,B 0.000,C 90.000,E1 225.810} C_DIS
LIN {X 0.010,Y -150.501,Z 1849.239,A 0.000,B 0.000,C 90.000,E1 223.095} C_DIS
LIN {X 0.040,Y -147.225,Z 1849.214,A 0.000,B 0.000,C 90.000,E1 218.543} C_DIS
LIN {X 0.010,Y -145.247,Z 1849.194,A 0.000,B 0.000,C 90.000,E1 214.898} C_DIS
LIN {X -0.074,Y -142.364,Z 1849.163,A 0.000,B 0.000,C 90.000,E1 209.411} C_DIS
LIN {X 0.047,Y -141.750,Z 1849.153,A 0.000,B 0.000,C 90.000,E1 207.513} C_DIS
LIN {X -0.027,Y -139.493,Z 1849.117,A 0.000,B 0.000,C 90.000,E1 201.046} C_DIS
LIN {X 0.009,Y -138.998,Z 1849.101,A 0.000,B 0.000,C 90.000,E1 198.236} C_DIS
LIN {X -0.033,Y -138.337,Z 1849.055,A 0.000,B 0.000,C 90.000,E1 189.849} C_DIS
LIN {X -0.012,Y -139.412,Z 1849.008,A 0.000,B 0.000,C 90.000,E1 181.432} C_DIS
LIN {X 0.042,Y -141.325,Z 1848.972,A 0.000,B 0.000,C 90.000,E1 174.894} C_DIS
LIN {X -0.001,Y -142.682,Z 1848.956,A 0.000,B 0.000,C 90.000,E1 172.129} C_DIS
LIN {X -0.021,Y -145.041,Z 1848.931,A 0.000,B 0.000,C 90.000,E1 167.521} C_DIS
LIN {X -0.024,Y -147.667,Z 1848.910,A 0.000,B 0.000,C 90.000,E1 163.850} C_DIS
LIN {X 0.012,Y -150.308,Z 1848.890,A 0.000,B 0.000,C 90.000,E1 160.188} C_DIS
LIN {X 0.022,Y -153.719,Z 1848.870,A 0.000,B 0.000,C 90.000,E1 156.561} C_DIS
LIN {X -0.064,Y -157.132,Z 1848.850,A 0.000,B 0.000,C 90.000,E1 152.999} C_DIS
LIN {X 0.011,Y -161.279,Z 1848.830,A 0.000,B 0.000,C 90.000,E1 149.410} C_DIS
LIN {X 0.029,Y -164.396,Z 1848.815,A 0.000,B 0.000,C 90.000,E1 146.755} C_DIS
LIN {X 0.026,Y -169.074,Z 1848.796,A 0.000,B 0.000,C 90.000,E1 143.256} C_DIS
LIN {X -0.023,Y -171.633,Z 1848.786,A 0.000,B 0.000,C 90.000,E1 141.537} C_DIS
LIN {X 0.024,Y -176.593,Z 1848.767,A 0.000,B 0.000,C 90.000,E1 138.081} C_DIS
LIN {X -0.104,Y -180.891,Z 1848.753,A 0.000,B 0.000,C 90.000,E1 135.567} C_DIS
LIN {X 0.018,Y -186.306,Z 1848.734,A 0.000,B 0.000,C 90.000,E1 132.162} C_DIS
LIN {X 0.084,Y -190.941,Z 1848.720,A 0.000,B 0.000,C 90.000,E1 129.644} C_DIS
LIN {X 0.005,Y -196.710,Z 1848.702,A 0.000,B 0.000,C 90.000,E1 126.377} C_DIS
LIN {X 0.035,Y -199.956,Z 1848.693,A 0.000,B 0.000,C 90.000,E1 124.739} C_DIS
LIN {X -0.073,Y -205.871,Z 1848.675,A 0.000,B 0.000,C 90.000,E1 121.544} C_DIS
LIN {X 0.019,Y -210.687,Z 1848.662,A 0.000,B 0.000,C 90.000,E1 119.127} C_DIS
LIN {X 0.019,Y -216.515,Z 1848.644,A 0.000,B 0.000,C 90.000,E1 115.976} C_DIS
LIN {X 0.125,Y -219.619,Z 1848.636,A 0.000,B 0.000,C 90.000,E1 114.387} C_DIS
LIN {X 0.094,Y -224.066,Z 1848.621,A 0.000,B 0.000,C 90.000,E1 111.844} C_DIS
LIN {X 0.087,Y -283.511,Z 1848.621,A 0.000,B 0.000,C 90.000,E1 111.844} C_DIS
LIN {X 0.026,Y -284.474,Z 1848.621,A 0.000,B 0.000,C 90.000,E1 111.844} C_DIS
LIN {X -0.002,Y -290.071,Z 1848.620,A 0.000,B 0.000,C 90.000,E1 111.589} C_DIS
LIN {X -0.032,Y -292.833,Z 1848.619,A 0.000,B 0.000,C 90.000,E1 111.334} C_DIS
LIN {X -0.041,Y -296.571,Z 1848.615,A 0.000,B 0.000,C 90.000,E1 110.791} C_DIS
LIN {X -0.049,Y -309.838,Z 1848.603,A 0.000,B 0.000,C 90.000,E1 108.471} C_DIS
LIN {X -0.040,Y -324.470,Z 1848.590,A 0.000,B 0.000,C 90.000,E1 106.205} C_DIS
LIN {X 0.023,Y -338.193,Z 1848.579,A 0.000,B 0.000,C 90.000,E1 104.300} C_DIS
LIN {X -0.151,Y -353.106,Z 1848.569,A 0.000,B 0.000,C 90.000,E1 102.479} C_DIS
LIN {X -0.014,Y -371.504,Z 1848.558,A 0.000,B 0.000,C 90.000,E1 100.423} C_DIS
LIN {X 0.008,Y -390.379,Z 1848.548,A 0.000,B 0.000,C 90.000,E1 98.568} C_DIS
LIN {X -0.034,Y -409.597,Z 1848.538,A 0.000,B 0.000,C 90.000,E1 96.891} C_DIS
LIN {X -0.182,Y -431.980,Z 1848.529,A 0.000,B 0.000,C 90.000,E1 95.163} C_DIS
LIN {X -0.024,Y -440.246,Z 1848.525,A 0.000,B 0.000,C 90.000,E1 94.531} C_DIS
LIN {X -0.228,Y -443.899,Z 1848.523,A 0.000,B 0.000,C 90.000,E1 94.131} C_DIS
LIN {X -0.028,Y -445.429,Z 1848.521,A 0.000,B 0.000,C 90.000,E1 93.841} C_DIS
LIN {X 0.141,Y -446.582,Z 1848.520,A 0.000,B 0.000,C 90.000,E1 93.555} C_DIS
LIN {X 0.094,Y -447.988,Z 1848.517,A 0.000,B 0.000,C 90.000,E1 93.037} C_DIS
LIN {X 0.029,Y -448.402,Z 1848.514,A 0.000,B 0.000,C 90.000,E1 92.522} C_DIS
LIN {X -0.024,Y -447.888,Z 1848.511,A 0.000,B 0.000,C 90.000,E1 92.007} C_DIS
LIN {X -0.062,Y -446.375,Z 1848.508,A 0.000,B 0.000,C 90.000,E1 91.489} C_DIS
LIN {X 0.135,Y -445.168,Z 1848.507,A 0.000,B 0.000,C 90.000,E1 91.203} C_DIS
LIN {X -0.097,Y -435.350,Z 1848.498,A 0.000,B 0.000,C 90.000,E1 89.656} C_DIS
LIN {X -0.048,Y -425.408,Z 1848.489,A 0.000,B 0.000,C 90.000,E1 88.051} C_DIS
LIN {X -0.075,Y -413.634,Z 1848.479,A 0.000,B 0.000,C 90.000,E1 86.159} C_DIS
LIN {X 0.108,Y -401.767,Z 1848.468,A 0.000,B 0.000,C 90.000,E1 84.204} C_DIS
LIN {X 0.087,Y -389.820,Z 1848.457,A 0.000,B 0.000,C 90.000,E1 82.243} C_DIS
LIN {X -0.131,Y -377.888,Z 1848.446,A 0.000,B 0.000,C 90.000,E1 80.274} C_DIS
LIN {X -0.148,Y -361.202,Z 1848.430,A 0.000,B 0.000,C 90.000,E1 77.353} C_DIS
LIN {X -0.066,Y -345.566,Z 1848.413,A 0.000,B 0.000,C 90.000,E1 74.338} C_DIS
LIN {X -0.026,Y -333.571,Z 1848.399,A 0.000,B 0.000,C 90.000,E1 71.873} C_DIS
LIN {X -0.168,Y -321.838,Z 1848.385,A 0.000,B 0.000,C 90.000,E1 69.390} C_DIS
LIN {X -0.040,Y -309.190,Z 1848.369,A 0.000,B 0.000,C 90.000,E1 66.485} C_DIS
LIN {X -0.068,Y -299.614,Z 1848.357,A 0.000,B 0.000,C 90.000,E1 64.204} C_DIS
LIN {X 0.070,Y -287.520,Z 1848.340,A 0.000,B 0.000,C 90.000,E1 61.179} C_DIS
LIN {X 0.116,Y -278.119,Z 1848.327,A 0.000,B 0.000,C 90.000,E1 58.791} C_DIS
LIN {X -0.126,Y -268.668,Z 1848.313,A 0.000,B 0.000,C 90.000,E1 56.421} C_DIS
LIN {X 0.039,Y -260.487,Z 1848.302,A 0.000,B 0.000,C 90.000,E1 54.276} C_DIS
LIN {X -0.017,Y -252.266,Z 1848.290,A 0.000,B 0.000,C 90.000,E1 52.145} C_DIS
LIN {X 0.045,Y -242.680,Z 1848.276,A 0.000,B 0.000,C 90.000,E1 49.585} C_DIS
LIN {X 0.067,Y -233.265,Z 1848.261,A 0.000,B 0.000,C 90.000,E1 46.986} C_DIS
LIN {X 0.117,Y -222.966,Z 1848.244,A 0.000,B 0.000,C 90.000,E1 43.947} C_DIS
LIN {X -0.073,Y -213.155,Z 1848.227,A 0.000,B 0.000,C 90.000,E1 40.906} C_DIS
LIN {X 0.007,Y -204.146,Z 1848.210,A 0.000,B 0.000,C 90.000,E1 37.729} C_DIS
LIN {X -0.030,Y -196.047,Z 1848.192,A 0.000,B 0.000,C 90.000,E1 34.532} C_DIS
LIN {X -0.001,Y -188.637,Z 1848.174,A 0.000,B 0.000,C 90.000,E1 31.258} C_DIS
LIN {X -0.003,Y -182.852,Z 1848.158,A 0.000,B 0.000,C 90.000,E1 28.409} C_DIS
LIN {X -0.024,Y -182.901,Z 1848.158,A 0.000,B 0.000,C 90.000,E1 28.409} C_DIS
LIN {X 0.022,Y -189.959,Z 1848.153,A 0.000,B 0.000,C 90.000,E1 27.590} C_DIS
LIN {X -0.007,Y -192.164,Z 1848.151,A 0.000,B 0.000,C 90.000,E1 27.257} C_DIS
LIN {X -0.027,Y -193.622,Z 1848.147,A 0.000,B 0.000,C 90.000,E1 26.437} C_DIS
LIN {X 0.054,Y -194.076,Z 1848.142,A 0.000,B 0.000,C 90.000,E1 25.591} C_DIS
LIN {X 0.058,Y -194.175,Z 1848.138,A 0.000,B 0.000,C 90.000,E1 24.771} C_DIS
LIN {X -0.004,Y -193.912,Z 1848.129,A 0.000,B 0.000,C 90.000,E1 23.153} C_DIS
LIN {X 0.045,Y -193.029,Z 1848.115,A 0.000,B 0.000,C 90.000,E1 20.684} C_DIS
LIN {X 0.044,Y -191.517,Z 1848.097,A 0.000,B 0.000,C 90.000,E1 17.402} C_DIS
LIN {X 0.008,Y -190.021,Z 1848.078,A 0.000,B 0.000,C 90.000,E1 14.120} C_DIS
LIN {X 0.096,Y -188.359,Z 1848.056,A 0.000,B 0.000,C 90.000,E1 9.962} C_DIS
LIN {X 0.071,Y -186.958,Z 1848.028,A 0.000,B 0.000,C 90.000,E1 4.992} C_DIS
LIN {X -0.034,Y -186.387,Z 1847.997,A 0.000,B 0.000,C 90.000,E1 359.542} C_DIS
LIN {X -0.031,Y -186.524,Z 1847.970,A 0.000,B 0.000,C 90.000,E1 354.546} C_DIS
LIN {X -0.035,Y -186.920,Z 1847.947,A 0.000,B 0.000,C 90.000,E1 350.387} C_DIS
LIN {X -0.060,Y -187.930,Z 1847.919,A 0.000,B 0.000,C 90.000,E1 345.408} C_DIS
LIN {X 0.078,Y -189.352,Z 1847.896,A 0.000,B 0.000,C 90.000,E1 341.221} C_DIS
LIN {X -0.053,Y -191.667,Z 1847.868,A 0.000,B 0.000,C 90.000,E1 336.305} C_DIS
LIN {X -0.078,Y -194.934,Z 1847.841,A 0.000,B 0.000,C 90.000,E1 331.385} C_DIS
LIN {X -0.038,Y -198.124,Z 1847.818,A 0.000,B 0.000,C 90.000,E1 327.296} C_DIS
LIN {X 0.094,Y -201.884,Z 1847.796,A 0.000,B 0.000,C 90.000,E1 323.210} C_DIS
LIN {X 0.017,Y -206.247,Z 1847.773,A 0.000,B 0.000,C 90.000,E1 319.218} C_DIS
LIN {X -0.046,Y -210.690,Z 1847.756,A 0.000,B 0.000,C 90.000,E1 316.053} C_DIS
LIN {X 0.105,Y -213.482,Z 1847.747,A 0.000,B 0.000,C 90.000,E1 314.433} C_DIS
LIN {X -0.015,Y -216.853,Z 1847.738,A 0.000,B 0.000,C 90.000,E1 312.894} C_DIS
LIN {X 0.077,Y -221.012,Z 1847.730,A 0.000,B 0.000,C 90.000,E1 311.310} C_DIS
LIN {X -0.004,Y -224.691,Z 1847.723,A 0.000,B 0.000,C 90.000,E1 310.172} C_DIS
LIN {X -0.059,Y -228.899,Z 1847.717,A 0.000,B 0.000,C 90.000,E1 309.036} C_DIS
LIN {X -0.085,Y -235.208,Z 1847.708,A 0.000,B 0.000,C 90.000,E1 307.523} C_DIS
LIN {X 0.132,Y -245.798,Z 1847.696,A 0.000,B 0.000,C 90.000,E1 305.231} C_DIS
LIN {X -0.073,Y -257.479,Z 1847.684,A 0.000,B 0.000,C 90.000,E1 303.086} C_DIS
LIN {X -0.162,Y -266.022,Z 1847.676,A 0.000,B 0.000,C 90.000,E1 301.671} C_DIS
LIN {X -0.093,Y -282.066,Z 1847.662,A 0.000,B 0.000,C 90.000,E1 299.205} C_DIS
LIN {X 0.087,Y -293.979,Z 1847.653,A 0.000,B 0.000,C 90.000,E1 297.462} C_DIS
LIN {X 0.080,Y -305.901,Z 1847.643,A 0.000,B 0.000,C 90.000,E1 295.796} C_DIS
LIN {X 0.179,Y -320.082,Z 1847.633,A 0.000,B 0.000,C 90.000,E1 293.823} C_DIS
LIN {X -0.111,Y -331.899,Z 1847.624,A 0.000,B 0.000,C 90.000,E1 292.280} C_DIS
LIN {X -0.092,Y -341.000,Z 1847.617,A 0.000,B 0.000,C 90.000,E1 291.025} C_DIS
LIN {X 0.119,Y -349.494,Z 1847.610,A 0.000,B 0.000,C 90.000,E1 289.758} C_DIS
LIN {X 0.082,Y -355.421,Z 1847.605,A 0.000,B 0.000,C 90.000,E1 288.852} C_DIS
LIN {X 0.162,Y -359.121,Z 1847.601,A 0.000,B 0.000,C 90.000,E1 288.236} C_DIS
LIN {X 0.099,Y -364.002,Z 1847.596,A 0.000,B 0.000,C 90.000,E1 287.347} C_DIS
LIN {X -0.154,Y -368.081,Z 1847.592,A 0.000,B 0.000,C 90.000,E1 286.496} C_DIS
LIN {X -0.128,Y -371.458,Z 1847.587,A 0.000,B 0.000,C 90.000,E1 285.607} C_DIS
LIN {X -0.058,Y -373.303,Z 1847.583,A 0.000,B 0.000,C 90.000,E1 285.009} C_DIS
LIN {X 0.017,Y -374.791,Z 1847.580,A 0.000,B 0.000,C 90.000,E1 284.411} C_DIS
LIN {X 0.011,Y -375.909,Z 1847.577,A 0.000,B 0.000,C 90.000,E1 283.828} C_DIS
LIN {X 0.018,Y -376.567,Z 1847.574,A 0.000,B 0.000,C 90.000,E1 283.244} C_DIS
LIN {X 0.115,Y -376.847,Z 1847.570,A 0.000,B 0.000,C 90.000,E1 282.647} C_DIS
LIN {X 0.134,Y -376.674,Z 1847.567,A 0.000,B 0.000,C 90.000,E1 282.063} C_DIS
LIN {X 0.154,Y -376.059,Z 1847.564,A 0.000,B 0.000,C 90.000,E1 281.478} C_DIS
LIN {X 0.174,Y -374.979,Z 1847.561,A 0.000,B 0.000,C 90.000,E1 280.894} C_DIS
LIN {X 0.188,Y -373.412,Z 1847.557,A 0.000,B 0.000,C 90.000,E1 280.310} C_DIS
LIN {X 0.132,Y -370.297,Z 1847.553,A 0.000,B 0.000,C 90.000,E1 279.443} C_DIS
LIN {X -0.037,Y -362.048,Z 1847.541,A 0.000,B 0.000,C 90.000,E1 277.409} C_DIS
LIN {X 0.160,Y -357.867,Z 1847.536,A 0.000,B 0.000,C 90.000,E1 276.486} C_DIS
LIN {X 0.022,Y -354.415,Z 1847.533,A 0.000,B 0.000,C 90.000,E1 275.910} C_DIS
LIN {X -0.133,Y -350.325,Z 1847.530,A 0.000,B 0.000,C 90.000,E1 275.334} C_DIS
LIN {X 0.039,Y -345.536,Z 1847.526,A 0.000,B 0.000,C 90.000,E1 274.702} C_DIS
LIN {X -0.130,Y -340.072,Z 1847.523,A 0.000,B 0.000,C 90.000,E1 274.131} C_DIS
LIN {X -0.099,Y -334.161,Z 1847.520,A 0.000,B 0.000,C 90.000,E1 273.555} C_DIS
LIN {X -0.147,Y -328.092,Z 1847.517,A 0.000,B 0.000,C 90.000,E1 273.037} C_DIS
LIN {X 0.036,Y -321.786,Z 1847.514,A 0.000,B 0.000,C 90.000,E1 272.522} C_DIS
LIN {X -0.144,Y -315.217,Z 1847.512,A 0.000,B 0.000,C 90.000,E1 272.121} C_DIS
LIN {X -0.024,Y -308.544,Z 1847.510,A 0.000,B 0.000,C 90.000,E1 271.718} C_DIS
LIN {X 0.048,Y -301.395,Z 1847.508,A 0.000,B 0.000,C 90.000,E1 271.375} C_DIS
LIN {X 0.136,Y -293.978,Z 1847.506,A 0.000,B 0.000,C 90.000,E1 271.088} C_DIS
LIN {X -0.050,Y -286.400,Z 1847.505,A 0.000,B 0.000,C 90.000,E1 270.917} C_DIS
LIN {X 0.115,Y -271.549,Z 1847.503,A 0.000,B 0.000,C 90.000,E1 270.573} C_DIS
LIN {X 0.061,Y -250.027,Z 1847.501,A 0.000,B 0.000,C 90.000,E1 270.172} C_DIS
LIN {X -0.013,Y -241.577,Z 1847.500,A 0.000,B 0.000,C 90.000,E1 270.057} C_DIS
LIN {X 0.029,Y -229.258,Z 1847.500,A 0.000,B 0.000,C 90.000,E1 269.943} C_DIS
LIN {X 0.003,Y -181.551,Z 1847.500,A 0.000,B 0.000,C 90.000,E1 269.943} C_DIS
LIN {X -0.022,Y -180.815,Z 1847.471,A 0.000,B 0.000,C 90.000,E1 264.837} C_DIS
LIN {X 0.055,Y -178.918,Z 1847.443,A 0.000,B 0.000,C 90.000,E1 259.746} C_DIS
LIN {X -0.036,Y -175.963,Z 1847.415,A 0.000,B 0.000,C 90.000,E1 254.685} C_DIS
LIN {X 0.080,Y -175.439,Z 1847.410,A 0.000,B 0.000,C 90.000,E1 253.795} C_DIS
LIN {X -0.079,Y -172.195,Z 1847.386,A 0.000,B 0.000,C 90.000,E1 249.571} C_DIS
LIN {X -0.101,Y -171.669,Z 1847.382,A 0.000,B 0.000,C 90.000,E1 248.720} C_DIS
LIN {X 0.042,Y -167.894,Z 1847.358,A 0.000,B 0.000,C 90.000,E1 244.357} C_DIS
LIN {X 0.057,Y -166.633,Z 1847.348,A 0.000,B 0.000,C 90.000,E1 242.615} C_DIS
LIN {X -0.035,Y -162.618,Z 1847.324,A 0.000,B 0.000,C 90.000,E1 238.280} C_DIS
LIN {X 0.024,Y -161.305,Z 1847.314,A 0.000,B 0.000,C 90.000,E1 236.501} C_DIS
LIN {X -0.066,Y -157.302,Z 1847.289,A 0.000,B 0.000,C 90.000,E1 232.110} C_DIS
LIN {X 0.087,Y -155.278,Z 1847.275,A 0.000,B 0.000,C 90.000,E1 229.380} C_DIS
LIN {X 0.015,Y -151.643,Z 1847.250,A 0.000,B 0.000,C 90.000,E1 224.919} C_DIS
LIN {X -0.048,Y -150.512,Z 1847.240,A 0.000,B 0.000,C 90.000,E1 223.137} C_DIS
LIN {X -0.025,Y -147.237,Z 1847.214,A 0.000,B 0.000,C 90.000,E1 218.588} C_DIS
LIN {X 0.060,Y -145.260,Z 1847.194,A 0.000,B 0.000,C 90.000,E1 214.898} C_DIS
LIN {X -0.024,Y -142.372,Z 1847.163,A 0.000,B 0.000,C 90.000,E1 209.411} C_DIS
LIN {X -0.029,Y -141.756,Z 1847.153,A 0.000,B 0.000,C 90.000,E1 207.564} C_DIS
LIN {X 0.022,Y -139.497,Z 1847.117,A 0.000,B 0.000,C 90.000,E1 201.046} C_DIS
LIN {X 0.058,Y -139.003,Z 1847.101,A 0.000,B 0.000,C 90.000,E1 198.236} C_DIS
LIN {X 0.015,Y -138.338,Z 1847.055,A 0.000,B 0.000,C 90.000,E1 189.849} C_DIS
LIN {X 0.037,Y -139.406,Z 1847.008,A 0.000,B 0.000,C 90.000,E1 181.432} C_DIS
LIN {X -0.050,Y -141.316,Z 1846.972,A 0.000,B 0.000,C 90.000,E1 174.951} C_DIS
LIN {X 0.049,Y -142.675,Z 1846.956,A 0.000,B 0.000,C 90.000,E1 172.129} C_DIS
LIN {X 0.029,Y -145.028,Z 1846.931,A 0.000,B 0.000,C 90.000,E1 167.521} C_DIS
LIN {X -0.014,Y -147.655,Z 1846.910,A 0.000,B 0.000,C 90.000,E1 163.866} C_DIS
LIN {X 0.062,Y -150.292,Z 1846.890,A 0.000,B 0.000,C 90.000,E1 160.188} C_DIS
LIN {X -0.066,Y -153.698,Z 1846.870,A 0.000,B 0.000,C 90.000,E1 156.613} C_DIS
LIN {X -0.011,Y -157.112,Z 1846.850,A 0.000,B 0.000,C 90.000,E1 152.999} C_DIS
LIN {X 0.065,Y -161.254,Z 1846.830,A 0.000,B 0.000,C 90.000,E1 149.410} C_DIS
LIN {X -0.007,Y -164.373,Z 1846.815,A 0.000,B 0.000,C 90.000,E1 146.786} C_DIS
LIN {X -0.021,Y -169.047,Z 1846.796,A 0.000,B 0.000,C 90.000,E1 143.290} C_DIS
LIN {X 0.032,Y -171.609,Z 1846.786,A 0.000,B 0.000,C 90.000,E1 141.537} C_DIS
LIN {X 0.080,Y -176.564,Z 1846.767,A 0.000,B 0.000,C 90.000,E1 138.081} C_DIS
LIN {X -0.045,Y -180.862,Z 1846.753,A 0.000,B 0.000,C 90.000,E1 135.567} C_DIS
LIN {X -0.063,Y -186.275,Z 1846.734,A 0.000,B 0.000,C 90.000,E1 132.204} C_DIS
LIN {X -0.003,Y -190.911,Z 1846.720,A 0.000,B 0.000,C 90.000,E1 129.688} C_DIS
LIN {X 0.065,Y -196.677,Z 1846.702,A 0.000,B 0.000,C 90.000,E1 126.377} C_DIS
LIN {X -0.018,Y -199.920,Z 1846.693,A 0.000,B 0.000,C 90.000,E1 124.771} C_DIS
LIN {X 0.013,Y -204.311,Z 1846.680,A 0.000,B 0.000,C 90.000,E1 122.339} C_DIS
LIN {X -0.022,Y -210.657,Z 1846.662,A 0.000,B 0.000,C 90.000,E1 119.155} C_DIS
LIN {X 0.082,Y -216.480,Z 1846.644,A 0.000,B 0.000,C 90.000,E1 115.976} C_DIS
LIN {X -0.101,Y -219.592,Z 1846.636,A 0.000,B 0.000,C 90.000,E1 114.463} C_DIS
LIN {X -0.099,Y -224.059,Z 1846.621,A 0.000,B 0.000,C 90.000,E1 111.897} C_DIS
LIN {X 0.106,Y -283.198,Z 1846.621,A 0.000,B 0.000,C 90.000,E1 111.844} C_DIS
LIN {X 0.095,Y -287.800,Z 1846.621,A 0.000,B 0.000,C 90.000,E1 111.716} C_DIS
LIN {X 0.081,Y -289.866,Z 1846.620,A 0.000,B 0.000,C 90.000,E1 111.589} C_DIS
LIN {X -0.053,Y -292.690,Z 1846.619,A 0.000,B 0.000,C 90.000,E1 111.354} C_DIS
LIN {X 0.095,Y -296.425,Z 1846.616,A 0.000,B 0.000,C 90.000,E1 110.791} C_DIS
LIN {X -0.008,Y -309.680,Z 1846.603,A 0.000,B 0.000,C 90.000,E1 108.489} C_DIS
LIN {X 0.102,Y -324.295,Z 1846.590,A 0.000,B 0.000,C 90.000,E1 106.205} C_DIS
LIN {X 0.168,Y -338.004,Z 1846.580,A 0.000,B 0.000,C 90.000,E1 104.300} C_DIS
LIN {X -0.003,Y -352.900,Z 1846.569,A 0.000,B 0.000,C 90.000,E1 102.479} C_DIS
LIN {X 0.060,Y -371.293,Z 1846.558,A 0.000,B 0.000,C 90.000,E1 100.433} C_DIS
LIN {X 0.142,Y -390.164,Z 1846.548,A 0.000,B 0.000,C 90.000,E1 98.568} C_DIS
LIN {X 0.095,Y -409.377,Z 1846.538,A 0.000,B 0.000,C 90.000,E1 96.891} C_DIS
LIN {X -0.059,Y -431.757,Z 1846.529,A 0.000,B 0.000,C 90.000,E1 95.163} C_DIS
LIN {X 0.095,Y -440.066,Z 1846.525,A 0.000,B 0.000,C 90.000,E1 94.531} C_DIS
LIN {X -0.069,Y -443.752,Z 1846.523,A 0.000,B 0.000,C 90.000,E1 94.131} C_DIS
LIN {X 0.130,Y -445.316,Z 1846.521,A 0.000,B 0.000,C 90.000,E1 93.841} C_DIS
LIN {X -0.146,Y -446.494,Z 1846.520,A 0.000,B 0.000,C 90.000,E1 93.612} C_DIS
LIN {X -0.195,Y -447.940,Z 1846.517,A 0.000,B 0.000,C 90.000,E1 93.094} C_DIS
LIN {X 0.187,Y -448.389,Z 1846.514,A 0.000,B 0.000,C 90.000,E1 92.522} C_DIS
LIN {X 0.133,Y -447.910,Z 1846.511,A 0.000,B 0.000,C 90.000,E1 92.007} C_DIS
LIN {X 0.096,Y -446.437,Z 1846.508,A 0.000,B 0.000,C 90.000,E1 91.489} C_DIS
LIN {X -0.154,Y -445.255,Z 1846.507,A 0.000,B 0.000,C 90.000,E1 91.260} C_DIS
LIN {X 0.058,Y -435.456,Z 1846.498,A 0.000,B 0.000,C 90.000,E1 89.656} C_DIS
LIN {X 0.105,Y -425.520,Z 1846.489,A 0.000,B 0.000,C 90.000,E1 88.051} C_DIS
LIN {X 0.076,Y -413.745,Z 1846.479,A 0.000,B 0.000,C 90.000,E1 86.159} C_DIS
LIN {X -0.142,Y -401.879,Z 1846.468,A 0.000,B 0.000,C 90.000,E1 84.261} C_DIS
LIN {X -0.152,Y -389.932,Z 1846.457,A 0.000,B 0.000,C 90.000,E1 82.299} C_DIS
LIN {X 0.014,Y -378.000,Z 1846.446,A 0.000,B 0.000,C 90.000,E1 80.274} C_DIS
LIN {X -0.007,Y -361.305,Z 1846.430,A 0.000,B 0.000,C 90.000,E1 77.353} C_DIS
LIN {X 0.073,Y -345.661,Z 1846.413,A 0.000,B 0.000,C 90.000,E1 74.338} C_DIS
LIN {X 0.110,Y -333.663,Z 1846.399,A 0.000,B 0.000,C 90.000,E1 71.873} C_DIS
LIN {X -0.035,Y -321.927,Z 1846.385,A 0.000,B 0.000,C 90.000,E1 69.390} C_DIS
LIN {X 0.091,Y -309.272,Z 1846.370,A 0.000,B 0.000,C 90.000,E1 66.485} C_DIS
LIN {X 0.060,Y -299.694,Z 1846.357,A 0.000,B 0.000,C 90.000,E1 64.204} C_DIS
LIN {X -0.057,Y -287.596,Z 1846.340,A 0.000,B 0.000,C 90.000,E1 61.229} C_DIS
LIN {X -0.143,Y -278.198,Z 1846.327,A 0.000,B 0.000,C 90.000,E1 58.869} C_DIS
LIN {X -0.007,Y -268.747,Z 1846.313,A 0.000,B 0.000,C 90.000,E1 56.421} C_DIS
LIN {X -0.054,Y -260.569,Z 1846.302,A 0.000,B 0.000,C 90.000,E1 54.322} C_DIS
LIN {X -0.100,Y -252.350,Z 1846.290,A 0.000,B 0.000,C 90.000,E1 52.190} C_DIS
LIN {X 0.001,Y -242.762,Z 1846.276,A 0.000,B 0.000,C 90.000,E1 49.622} C_DIS
LIN {X 0.018,Y -233.345,Z 1846.261,A 0.000,B 0.000,C 90.000,E1 47.025} C_DIS
LIN {X -0.090,Y -223.040,Z 1846.245,A 0.000,B 0.000,C 90.000,E1 44.028} C_DIS
LIN {X 0.031,Y -213.224,Z 1846.227,A 0.000,B 0.000,C 90.000,E1 40.906} C_DIS
LIN {X 0.110,Y -204.209,Z 1846.210,A 0.000,B 0.000,C 90.000,E1 37.729} C_DIS
LIN {X 0.070,Y -196.107,Z 1846.192,A 0.000,B 0.000,C 90.000,E1 34.532} C_DIS
LIN {X -0.019,Y -188.514,Z 1846.173,A 0.000,B 0.000,C 90.000,E1 31.209} C_DIS
LIN {X -0.040,Y -188.530,Z 1846.173,A 0.000,B 0.000,C 90.000,E1 31.209} C_DIS
LIN {X 0.066,Y -197.038,Z 1846.167,A 0.000,B 0.000,C 90.000,E1 30.079} C_DIS
LIN {X -0.038,Y -198.123,Z 1846.165,A 0.000,B 0.000,C 90.000,E1 29.745} C_DIS
LIN {X -0.096,Y -199.001,Z 1846.161,A 0.000,B 0.000,C 90.000,E1 28.949} C_DIS
LIN {X 0.026,Y -199.181,Z 1846.156,A 0.000,B 0.000,C 90.000,E1 28.103} C_DIS
LIN {X -0.024,Y -199.057,Z 1846.152,A 0.000,B 0.000,C 90.000,E1 27.308} C_DIS
LIN {X 0.052,Y -198.351,Z 1846.143,A 0.000,B 0.000,C 90.000,E1 25.668} C_DIS
LIN {X -0.025,Y -196.888,Z 1846.129,A 0.000,B 0.000,C 90.000,E1 23.259} C_DIS
LIN {X 0.015,Y -194.811,Z 1846.111,A 0.000,B 0.000,C 90.000,E1 19.993} C_DIS
LIN {X 0.034,Y -192.301,Z 1846.088,A 0.000,B 0.000,C 90.000,E1 15.898} C_DIS
LIN {X 0.087,Y -190.059,Z 1846.066,A 0.000,B 0.000,C 90.000,E1 11.771} C_DIS
LIN {X 0.012,Y -187.998,Z 1846.038,A 0.000,B 0.000,C 90.000,E1 6.834} C_DIS
LIN {X -0.020,Y -186.684,Z 1846.006,A 0.000,B 0.000,C 90.000,E1 1.031} C_DIS
LIN {X -0.046,Y -186.321,Z 1845.979,A 0.000,B 0.000,C 90.000,E1 356.216} C_DIS
LIN {X -0.010,Y -186.377,Z 1845.960,A 0.000,B 0.000,C 90.000,E1 352.875} C_DIS
LIN {X -0.049,Y -187.153,Z 1845.928,A 0.000,B 0.000,C 90.000,E1 347.061} C_DIS
LIN {X 0.033,Y -188.713,Z 1845.900,A 0.000,B 0.000,C 90.000,E1 342.054} C_DIS
LIN {X -0.003,Y -190.930,Z 1845.873,A 0.000,B 0.000,C 90.000,E1 337.102} C_DIS
LIN {X 0.042,Y -194.050,Z 1845.845,A 0.000,B 0.000,C 90.000,E1 332.153} C_DIS
LIN {X 0.024,Y -197.207,Z 1845.823,A 0.000,B 0.000,C 90.000,E1 328.074} C_DIS
LIN {X -0.040,Y -200.888,Z 1845.800,A 0.000,B 0.000,C 90.000,E1 324.036} C_DIS
LIN {X 0.046,Y -205.134,Z 1845.778,A 0.000,B 0.000,C 90.000,E1 319.989} C_DIS
LIN {X -0.046,Y -209.354,Z 1845.760,A 0.000,B 0.000,C 90.000,E1 316.824} C_DIS
LIN {X -0.059,Y -211.963,Z 1845.751,A 0.000,B 0.000,C 90.000,E1 315.243} C_DIS
LIN {X 0.108,Y -215.097,Z 1845.743,A 0.000,B 0.000,C 90.000,E1 313.623} C_DIS
LIN {X 0.018,Y -218.899,Z 1845.734,A 0.000,B 0.000,C 90.000,E1 312.081} C_DIS
LIN {X -0.015,Y -223.509,Z 1845.725,A 0.000,B 0.000,C 90.000,E1 310.539} C_DIS
LIN {X 0.036,Y -229.078,Z 1845.717,A 0.000,B 0.000,C 90.000,E1 308.991} C_DIS
LIN {X -0.025,Y -235.415,Z 1845.708,A 0.000,B 0.000,C 90.000,E1 307.488} C_DIS
LIN {X 0.050,Y -246.060,Z 1845.696,A 0.000,B 0.000,C 90.000,E1 305.231} C_DIS
LIN {X 0.088,Y -259.866,Z 1845.682,A 0.000,B 0.000,C 90.000,E1 302.673} C_DIS
LIN {X -0.048,Y -277.822,Z 1845.666,A 0.000,B 0.000,C 90.000,E1 299.873} C_DIS
LIN {X 0.016,Y -294.413,Z 1845.653,A 0.000,B 0.000,C 90.000,E1 297.462} C_DIS
LIN {X 0.012,Y -306.377,Z 1845.643,A 0.000,B 0.000,C 90.000,E1 295.796} C_DIS
LIN {X 0.118,Y -320.613,Z 1845.632,A 0.000,B 0.000,C 90.000,E1 293.823} C_DIS
LIN {X -0.041,Y -332.482,Z 1845.624,A 0.000,B 0.000,C 90.000,E1 292.259} C_DIS
LIN {X 0.177,Y -341.627,Z 1845.617,A 0.000,B 0.000,C 90.000,E1 290.972} C_DIS
LIN {X 0.076,Y -350.132,Z 1845.610,A 0.000,B 0.000,C 90.000,E1 289.758} C_DIS
LIN {X 0.045,Y -356.102,Z 1845.605,A 0.000,B 0.000,C 90.000,E1 288.852} C_DIS
LIN {X 0.065,Y -361.498,Z 1845.600,A 0.000,B 0.000,C 90.000,E1 287.946} C_DIS
LIN {X 0.140,Y -366.104,Z 1845.595,A 0.000,B 0.000,C 90.000,E1 287.040} C_DIS
LIN {X -0.206,Y -369.909,Z 1845.590,A 0.000,B 0.000,C 90.000,E1 286.205} C_DIS
LIN {X -0.145,Y -372.075,Z 1845.587,A 0.000,B 0.000,C 90.000,E1 285.607} C_DIS
LIN {X -0.070,Y -373.913,Z 1845.583,A 0.000,B 0.000,C 90.000,E1 285.009} C_DIS
LIN {X 0.008,Y -375.372,Z 1845.580,A 0.000,B 0.000,C 90.000,E1 284.411} C_DIS
LIN {X 0.006,Y -376.457,Z 1845.577,A 0.000,B 0.000,C 90.000,E1 283.828} C_DIS
LIN {X 0.016,Y -377.105,Z 1845.574,A 0.000,B 0.000,C 90.000,E1 283.244} C_DIS
LIN {X 0.118,Y -377.331,Z 1845.570,A 0.000,B 0.000,C 90.000,E1 282.647} C_DIS
LIN {X 0.139,Y -377.141,Z 1845.567,A 0.000,B 0.000,C 90.000,E1 282.063} C_DIS
LIN {X 0.163,Y -376.475,Z 1845.564,A 0.000,B 0.000,C 90.000,E1 281.478} C_DIS
LIN {X 0.185,Y -375.366,Z 1845.561,A 0.000,B 0.000,C 90.000,E1 280.894} C_DIS
LIN {X -0.166,Y -373.764,Z 1845.557,A 0.000,B 0.000,C 90.000,E1 280.366} C_DIS
LIN {X 0.210,Y -371.769,Z 1845.554,A 0.000,B 0.000,C 90.000,E1 279.726} C_DIS
LIN {X 0.012,Y -363.541,Z 1845.543,A 0.000,B 0.000,C 90.000,E1 277.701} C_DIS
LIN {X -0.094,Y -360.989,Z 1845.540,A 0.000,B 0.000,C 90.000,E1 277.125} C_DIS
LIN {X 0.101,Y -356.471,Z 1845.535,A 0.000,B 0.000,C 90.000,E1 276.201} C_DIS
LIN {X -0.042,Y -352.720,Z 1845.531,A 0.000,B 0.000,C 90.000,E1 275.625} C_DIS
LIN {X 0.144,Y -348.254,Z 1845.528,A 0.000,B 0.000,C 90.000,E1 274.992} C_DIS
LIN {X -0.041,Y -343.090,Z 1845.525,A 0.000,B 0.000,C 90.000,E1 274.416} C_DIS
LIN {X 0.113,Y -337.151,Z 1845.521,A 0.000,B 0.000,C 90.000,E1 273.784} C_DIS
LIN {X -0.086,Y -331.092,Z 1845.518,A 0.000,B 0.000,C 90.000,E1 273.269} C_DIS
LIN {X 0.011,Y -324.937,Z 1845.515,A 0.000,B 0.000,C 90.000,E1 272.751} C_DIS
LIN {X 0.002,Y -318.397,Z 1845.513,A 0.000,B 0.000,C 90.000,E1 272.293} C_DIS
LIN {X -0.013,Y -311.775,Z 1845.510,A 0.000,B 0.000,C 90.000,E1 271.892} C_DIS
LIN {X -0.075,Y -304.854,Z 1845.509,A 0.000,B 0.000,C 90.000,E1 271.547} C_DIS
LIN {X -0.135,Y -297.502,Z 1845.507,A 0.000,B 0.000,C 90.000,E1 271.260} C_DIS
LIN {X 0.107,Y -289.775,Z 1845.505,A 0.000,B 0.000,C 90.000,E1 270.974} C_DIS
LIN {X -0.029,Y -278.607,Z 1845.504,A 0.000,B 0.000,C 90.000,E1 270.745} C_DIS
LIN {X 0.094,Y -253.245,Z 1845.501,A 0.000,B 0.000,C 90.000,E1 270.229} C_DIS
LIN {X 0.000,Y -245.560,Z 1845.501,A 0.000,B 0.000,C 90.000,E1 270.115} C_DIS
LIN {X -0.047,Y -234.936,Z 1845.500,A 0.000,B 0.000,C 90.000,E1 270.000} C_DIS
LIN {X 0.052,Y -226.769,Z 1845.500,A 0.000,B 0.000,C 90.000,E1 269.943} C_DIS
LIN {X 0.021,Y -181.552,Z 1845.500,A 0.000,B 0.000,C 90.000,E1 269.943} C_DIS
LIN {X -0.021,Y -180.815,Z 1845.471,A 0.000,B 0.000,C 90.000,E1 264.837} C_DIS
LIN {X 0.056,Y -178.917,Z 1845.443,A 0.000,B 0.000,C 90.000,E1 259.746} C_DIS
LIN {X -0.035,Y -175.963,Z 1845.415,A 0.000,B 0.000,C 90.000,E1 254.685} C_DIS
LIN {X 0.081,Y -175.439,Z 1845.410,A 0.000,B 0.000,C 90.000,E1 253.795} C_DIS
LIN {X -0.078,Y -172.196,Z 1845.386,A 0.000,B 0.000,C 90.000,E1 249.571} C_DIS
LIN {X -0.100,Y -171.669,Z 1845.382,A 0.000,B 0.000,C 90.000,E1 248.720} C_DIS
LIN {X 0.043,Y -167.895,Z 1845.358,A 0.000,B 0.000,C 90.000,E1 244.357} C_DIS
LIN {X 0.059,Y -166.634,Z 1845.348,A 0.000,B 0.000,C 90.000,E1 242.615} C_DIS
LIN {X -0.034,Y -162.619,Z 1845.324,A 0.000,B 0.000,C 90.000,E1 238.280} C_DIS
LIN {X 0.025,Y -161.305,Z 1845.314,A 0.000,B 0.000,C 90.000,E1 236.501} C_DIS
LIN {X -0.065,Y -157.302,Z 1845.289,A 0.000,B 0.000,C 90.000,E1 232.110} C_DIS
LIN {X 0.087,Y -155.278,Z 1845.275,A 0.000,B 0.000,C 90.000,E1 229.380} C_DIS
LIN {X 0.016,Y -151.644,Z 1845.250,A 0.000,B 0.000,C 90.000,E1 224.919} C_DIS
LIN {X -0.047,Y -150.512,Z 1845.240,A 0.000,B 0.000,C 90.000,E1 223.137} C_DIS
LIN {X -0.024,Y -147.237,Z 1845.214,A 0.000,B 0.000,C 90.000,E1 218.588} C_DIS
LIN {X 0.060,Y -145.261,Z 1845.194,A 0.000,B 0.000,C 90.000,E1 214.898} C_DIS
LIN {X -0.024,Y -142.372,Z 1845.163,A 0.000,B 0.000,C 90.000,E1 209.411} C_DIS
LIN {X -0.028,Y -141.757,Z 1845.153,A 0.000,B 0.000,C 90.000,E1 207.564} C_DIS
LIN {X 0.023,Y -139.498,Z 1845.117,A 0.000,B 0.000,C 90.000,E1 201.046} C_DIS
LIN {X 0.059,Y -139.004,Z 1845.101,A 0.000,B 0.000,C 90.000,E1 198.236} C_DIS
LIN {X 0.016,Y -138.338,Z 1845.055,A 0.000,B 0.000,C 90.000,E1 189.849} C_DIS
LIN {X 0.038,Y -139.406,Z 1845.008,A 0.000,B 0.000,C 90.000,E1 181.432} C_DIS
LIN {X -0.048,Y -141.316,Z 1844.972,A 0.000,B 0.000,C 90.000,E1 174.951} C_DIS
LIN {X 0.050,Y -142.674,Z 1844.956,A 0.000,B 0.000,C 90.000,E1 172.129} C_DIS
LIN {X 0.030,Y -145.028,Z 1844.931,A 0.000,B 0.000,C 90.000,E1 167.521} C_DIS
LIN {X -0.013,Y -147.654,Z 1844.910,A 0.000,B 0.000,C 90.000,E1 163.866} C_DIS
LIN {X 0.064,Y -150.291,Z 1844.890,A 0.000,B 0.000,C 90.000,E1 160.188} C_DIS
LIN {X -0.066,Y -153.698,Z 1844.870,A 0.000,B 0.000,C 90.000,E1 156.613} C_DIS
LIN {X -0.010,Y -157.112,Z 1844.850,A 0.000,B 0.000,C 90.000,E1 152.999} C_DIS
LIN {X 0.066,Y -161.254,Z 1844.830,A 0.000,B 0.000,C 90.000,E1 149.410} C_DIS
LIN {X -0.006,Y -164.373,Z 1844.815,A 0.000,B 0.000,C 90.000,E1 146.786} C_DIS
LIN {X -0.019,Y -169.046,Z 1844.796,A 0.000,B 0.000,C 90.000,E1 143.290} C_DIS
LIN {X 0.034,Y -171.608,Z 1844.786,A 0.000,B 0.000,C 90.000,E1 141.537} C_DIS
LIN {X 0.081,Y -176.563,Z 1844.767,A 0.000,B 0.000,C 90.000,E1 138.081} C_DIS
LIN {X -0.045,Y -180.862,Z 1844.753,A 0.000,B 0.000,C 90.000,E1 135.567} C_DIS
LIN {X -0.060,Y -186.274,Z 1844.734,A 0.000,B 0.000,C 90.000,E1 132.204} C_DIS
LIN {X -0.002,Y -190.909,Z 1844.720,A 0.000,B 0.000,C 90.000,E1 129.688} C_DIS
LIN {X 0.066,Y -196.676,Z 1844.702,A 0.000,B 0.000,C 90.000,E1 126.377} C_DIS
LIN {X -0.016,Y -199.919,Z 1844.693,A 0.000,B 0.000,C 90.000,E1 124.771} C_DIS
LIN {X 0.015,Y -204.311,Z 1844.680,A 0.000,B 0.000,C 90.000,E1 122.339} C_DIS
LIN {X -0.021,Y -210.657,Z 1844.662,A 0.000,B 0.000,C 90.000,E1 119.155} C_DIS
LIN {X 0.084,Y -216.479,Z 1844.644,A 0.000,B 0.000,C 90.000,E1 115.976} C_DIS
LIN {X -0.100,Y -219.592,Z 1844.636,A 0.000,B 0.000,C 90.000,E1 114.463} C_DIS
LIN {X -0.098,Y -224.058,Z 1844.621,A 0.000,B 0.000,C 90.000,E1 111.897} C_DIS
LIN {X 0.108,Y -283.386,Z 1844.621,A 0.000,B 0.000,C 90.000,E1 111.844} C_DIS
LIN {X 0.096,Y -287.815,Z 1844.621,A 0.000,B 0.000,C 90.000,E1 111.716} C_DIS
LIN {X 0.083,Y -289.872,Z 1844.620,A 0.000,B 0.000,C 90.000,E1 111.589} C_DIS
LIN {X -0.052,Y -292.691,Z 1844.619,A 0.000,B 0.000,C 90.000,E1 111.354} C_DIS
LIN {X 0.093,Y -296.427,Z 1844.616,A 0.000,B 0.000,C 90.000,E1 110.791} C_DIS
LIN {X -0.010,Y -309.682,Z 1844.603,A 0.000,B 0.000,C 90.000,E1 108.489} C_DIS
LIN {X 0.100,Y -324.297,Z 1844.590,A 0.000,B 0.000,C 90.000,E1 106.205} C_DIS
LIN {X 0.165,Y -338.006,Z 1844.580,A 0.000,B 0.000,C 90.000,E1 104.300} C_DIS
LIN {X -0.006,Y -352.902,Z 1844.569,A 0.000,B 0.000,C 90.000,E1 102.479} C_DIS
LIN {X 0.056,Y -371.296,Z 1844.558,A 0.000,B 0.000,C 90.000,E1 100.433} C_DIS
LIN {X 0.140,Y -390.168,Z 1844.548,A 0.000,B 0.000,C 90.000,E1 98.568} C_DIS
LIN {X 0.092,Y -409.381,Z 1844.538,A 0.000,B 0.000,C 90.000,E1 96.891} C_DIS
LIN {X -0.061,Y -431.759,Z 1844.529,A 0.000,B 0.000,C 90.000,E1 95.163} C_DIS
LIN {X 0.094,Y -440.064,Z 1844.525,A 0.000,B 0.000,C 90.000,E1 94.531} C_DIS
LIN {X -0.075,Y -443.748,Z 1844.523,A 0.000,B 0.000,C 90.000,E1 94.131} C_DIS
LIN {X 0.125,Y -445.309,Z 1844.521,A 0.000,B 0.000,C 90.000,E1 93.841} C_DIS
LIN {X -0.151,Y -446.485,Z 1844.520,A 0.000,B 0.000,C 90.000,E1 93.612} C_DIS
LIN {X -0.200,Y -447.929,Z 1844.517,A 0.000,B 0.000,C 90.000,E1 93.094} C_DIS
LIN {X 0.182,Y -448.374,Z 1844.514,A 0.000,B 0.000,C 90.000,E1 92.522} C_DIS
LIN {X 0.128,Y -447.893,Z 1844.511,A 0.000,B 0.000,C 90.000,E1 92.007} C_DIS
LIN {X 0.090,Y -446.417,Z 1844.508,A 0.000,B 0.000,C 90.000,E1 91.489} C_DIS
LIN {X -0.160,Y -445.233,Z 1844.507,A 0.000,B 0.000,C 90.000,E1 91.260} C_DIS
LIN {X 0.052,Y -435.432,Z 1844.498,A 0.000,B 0.000,C 90.000,E1 89.656} C_DIS
LIN {X 0.098,Y -425.497,Z 1844.489,A 0.000,B 0.000,C 90.000,E1 88.051} C_DIS
LIN {X 0.070,Y -413.722,Z 1844.479,A 0.000,B 0.000,C 90.000,E1 86.159} C_DIS
LIN {X -0.149,Y -401.853,Z 1844.468,A 0.000,B 0.000,C 90.000,E1 84.261} C_DIS
LIN {X -0.159,Y -389.908,Z 1844.457,A 0.000,B 0.000,C 90.000,E1 82.299} C_DIS
LIN {X 0.006,Y -377.975,Z 1844.446,A 0.000,B 0.000,C 90.000,E1 80.274} C_DIS
LIN {X -0.014,Y -361.280,Z 1844.430,A 0.000,B 0.000,C 90.000,E1 77.353} C_DIS
LIN {X 0.064,Y -345.635,Z 1844.413,A 0.000,B 0.000,C 90.000,E1 74.338} C_DIS
LIN {X 0.101,Y -333.638,Z 1844.399,A 0.000,B 0.000,C 90.000,E1 71.873} C_DIS
LIN {X -0.043,Y -321.899,Z 1844.385,A 0.000,B 0.000,C 90.000,E1 69.390} C_DIS
LIN {X 0.082,Y -309.244,Z 1844.370,A 0.000,B 0.000,C 90.000,E1 66.485} C_DIS
LIN {X 0.051,Y -299.663,Z 1844.357,A 0.000,B 0.000,C 90.000,E1 64.204} C_DIS
LIN {X 0.185,Y -287.565,Z 1844.340,A 0.000,B 0.000,C 90.000,E1 61.179} C_DIS
LIN {X -0.154,Y -278.168,Z 1844.327,A 0.000,B 0.000,C 90.000,E1 58.869} C_DIS
LIN {X -0.017,Y -268.719,Z 1844.313,A 0.000,B 0.000,C 90.000,E1 56.421} C_DIS
LIN {X -0.065,Y -260.542,Z 1844.302,A 0.000,B 0.000,C 90.000,E1 54.322} C_DIS
LIN {X -0.111,Y -252.323,Z 1844.290,A 0.000,B 0.000,C 90.000,E1 52.190} C_DIS
LIN {X -0.010,Y -242.735,Z 1844.276,A 0.000,B 0.000,C 90.000,E1 49.622} C_DIS
LIN {X 0.007,Y -233.317,Z 1844.261,A 0.000,B 0.000,C 90.000,E1 47.025} C_DIS
LIN {X -0.102,Y -223.013,Z 1844.245,A 0.000,B 0.000,C 90.000,E1 44.028} C_DIS
LIN {X 0.020,Y -213.199,Z 1844.227,A 0.000,B 0.000,C 90.000,E1 40.906} C_DIS
LIN {X 0.098,Y -204.187,Z 1844.210,A 0.000,B 0.000,C 90.000,E1 37.729} C_DIS
LIN {X 0.058,Y -196.090,Z 1844.192,A 0.000,B 0.000,C 90.000,E1 34.532} C_DIS
LIN {X 0.000,Y -194.462,Z 1844.188,A 0.000,B 0.000,C 90.000,E1 33.865} C_DIS
LIN {X -0.022,Y -194.505,Z 1844.188,A 0.000,B 0.000,C 90.000,E1 33.865} C_DIS
LIN {X -0.087,Y -201.196,Z 1844.183,A 0.000,B 0.000,C 90.000,E1 32.959} C_DIS
LIN {X 0.011,Y -203.299,Z 1844.181,A 0.000,B 0.000,C 90.000,E1 32.546} C_DIS
LIN {X 0.111,Y -204.069,Z 1844.179,A 0.000,B 0.000,C 90.000,E1 32.133} C_DIS
LIN {X 0.090,Y -204.624,Z 1844.174,A 0.000,B 0.000,C 90.000,E1 31.337} C_DIS
LIN {X 0.075,Y -204.612,Z 1844.170,A 0.000,B 0.000,C 90.000,E1 30.541} C_DIS
LIN {X 0.051,Y -203.867,Z 1844.161,A 0.000,B 0.000,C 90.000,E1 28.949} C_DIS
LIN {X -0.079,Y -202.680,Z 1844.152,A 0.000,B 0.000,C 90.000,E1 27.385} C_DIS
LIN {X -0.020,Y -199.851,Z 1844.134,A 0.000,B 0.000,C 90.000,E1 24.155} C_DIS
LIN {X -0.055,Y -196.510,Z 1844.112,A 0.000,B 0.000,C 90.000,E1 20.120} C_DIS
LIN {X 0.073,Y -192.969,Z 1844.084,A 0.000,B 0.000,C 90.000,E1 15.190} C_DIS
LIN {X 0.093,Y -189.993,Z 1844.057,A 0.000,B 0.000,C 90.000,E1 10.254} C_DIS
LIN {X 0.059,Y -187.545,Z 1844.025,A 0.000,B 0.000,C 90.000,E1 4.473} C_DIS
LIN {X -0.034,Y -186.434,Z 1843.997,A 0.000,B 0.000,C 90.000,E1 359.542} C_DIS
LIN {X -0.036,Y -185.978,Z 1843.970,A 0.000,B 0.000,C 90.000,E1 354.546} C_DIS
LIN {X 0.006,Y -186.438,Z 1843.937,A 0.000,B 0.000,C 90.000,E1 348.701} C_DIS
LIN {X -0.078,Y -188.094,Z 1843.905,A 0.000,B 0.000,C 90.000,E1 342.906} C_DIS
